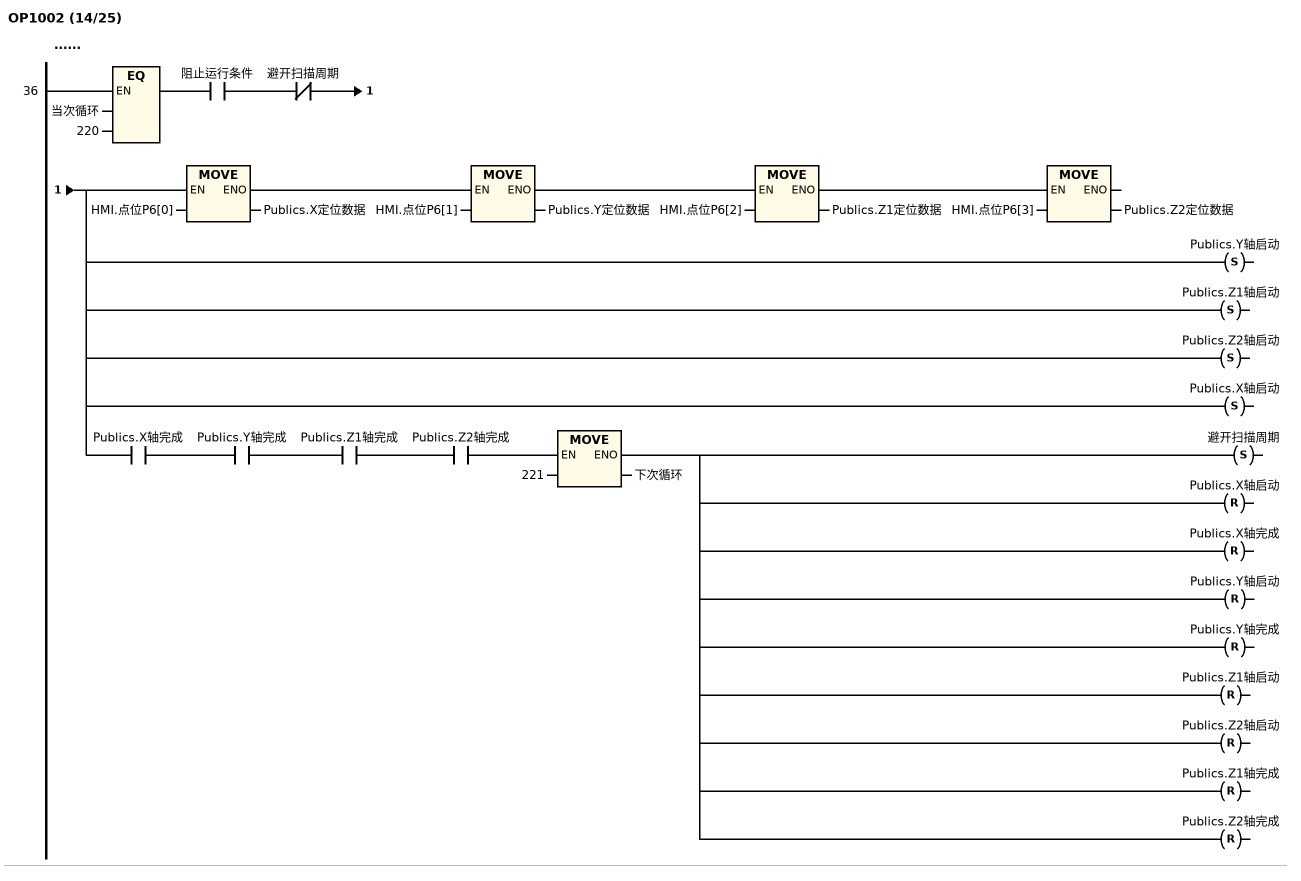
// NETWORK 36: ......
_w44 := 当次循环 = 220 AND 阻止运行条件 AND NOT 避开扫描周期;
IF _w44 THEN Publics.X定位数据 := HMI.点位P6[0]; END_IF
IF _w44 THEN Publics.Y定位数据 := HMI.点位P6[1]; END_IF
IF _w44 THEN Publics.Z1定位数据 := HMI.点位P6[2]; END_IF
IF _w44 THEN Publics.Z2定位数据 := HMI.点位P6[3]; END_IF
Publics.Y轴启动 S= _w44;
Publics.Z1轴启动 S= _w44;
Publics.Z2轴启动 S= _w44;
Publics.X轴启动 S= _w44;
IF _w44 AND Publics.X轴完成 AND Publics.Y轴完成 AND Publics.Z1轴完成 AND Publics.Z2轴完成 THEN 下次循环 := 221; END_IF
_w45 := _w44 AND Publics.X轴完成 AND Publics.Y轴完成 AND Publics.Z1轴完成 AND Publics.Z2轴完成;
避开扫描周期 S= _w45;
Publics.X轴启动 R= _w45;
Publics.X轴完成 R= _w45;
Publics.Y轴启动 R= _w45;
Publics.Y轴完成 R= _w45;
Publics.Z1轴启动 R= _w45;
Publics.Z2轴启动 R= _w45;
Publics.Z1轴完成 R= _w45;
Publics.Z2轴完成 R= _w45;

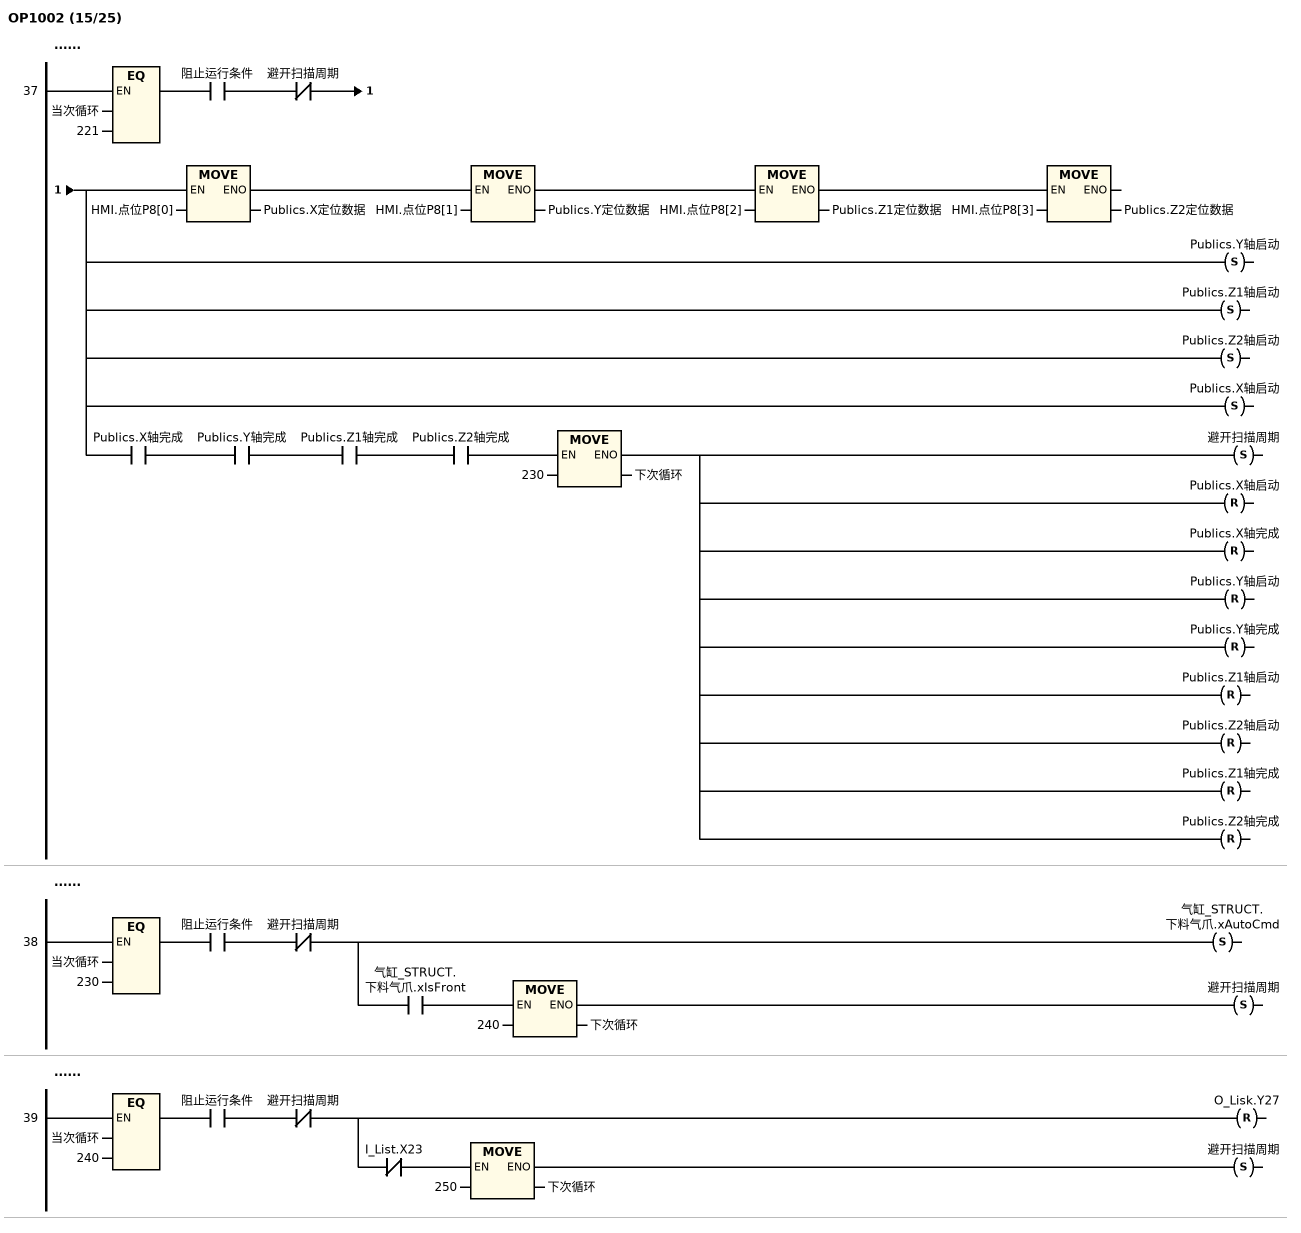
// NETWORK 37: ......
_w46 := 当次循环 = 221 AND 阻止运行条件 AND NOT 避开扫描周期;
IF _w46 THEN Publics.X定位数据 := HMI.点位P8[0]; END_IF
IF _w46 THEN Publics.Y定位数据 := HMI.点位P8[1]; END_IF
IF _w46 THEN Publics.Z1定位数据 := HMI.点位P8[2]; END_IF
IF _w46 THEN Publics.Z2定位数据 := HMI.点位P8[3]; END_IF
Publics.Y轴启动 S= _w46;
Publics.Z1轴启动 S= _w46;
Publics.Z2轴启动 S= _w46;
Publics.X轴启动 S= _w46;
IF _w46 AND Publics.X轴完成 AND Publics.Y轴完成 AND Publics.Z1轴完成 AND Publics.Z2轴完成 THEN 下次循环 := 230; END_IF
_w47 := _w46 AND Publics.X轴完成 AND Publics.Y轴完成 AND Publics.Z1轴完成 AND Publics.Z2轴完成;
避开扫描周期 S= _w47;
Publics.X轴启动 R= _w47;
Publics.X轴完成 R= _w47;
Publics.Y轴启动 R= _w47;
Publics.Y轴完成 R= _w47;
Publics.Z1轴启动 R= _w47;
Publics.Z2轴启动 R= _w47;
Publics.Z1轴完成 R= _w47;
Publics.Z2轴完成 R= _w47;

// NETWORK 38: ......
_w48 := 当次循环 = 230 AND 阻止运行条件 AND NOT 避开扫描周期;
气缸_STRUCT.下料气爪.xAutoCmd S= _w48;
IF _w48 AND 气缸_STRUCT.下料气爪.xIsFront THEN 下次循环 := 240; END_IF
避开扫描周期 S= _w48 AND 气缸_STRUCT.下料气爪.xIsFront;

// NETWORK 39: ......
_w49 := 当次循环 = 240 AND 阻止运行条件 AND NOT 避开扫描周期;
O_Lisk.Y27 R= _w49;
IF _w49 AND NOT I_List.X23 THEN 下次循环 := 250; END_IF
避开扫描周期 S= _w49 AND NOT I_List.X23;

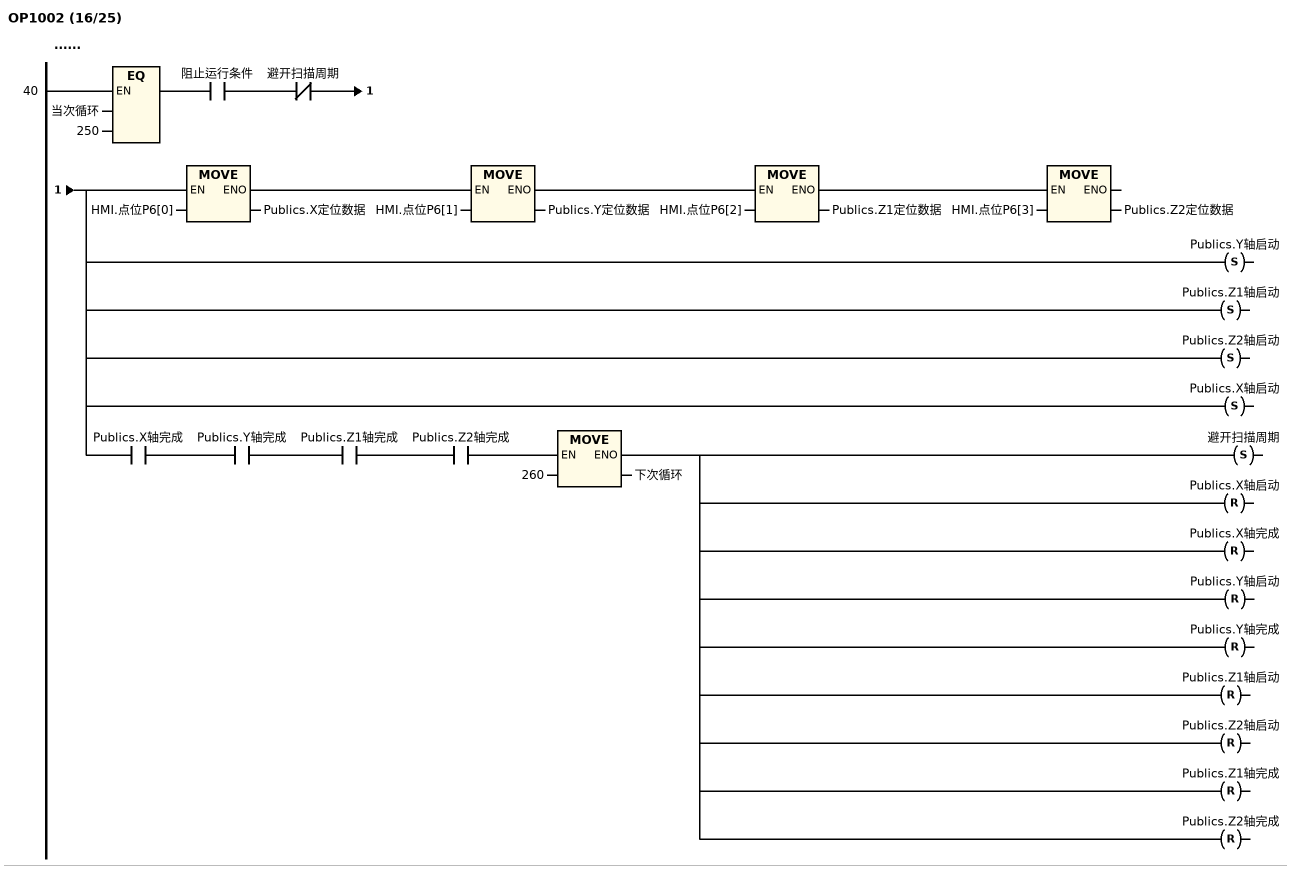
// NETWORK 40: ......
_w50 := 当次循环 = 250 AND 阻止运行条件 AND NOT 避开扫描周期;
IF _w50 THEN Publics.X定位数据 := HMI.点位P6[0]; END_IF
IF _w50 THEN Publics.Y定位数据 := HMI.点位P6[1]; END_IF
IF _w50 THEN Publics.Z1定位数据 := HMI.点位P6[2]; END_IF
IF _w50 THEN Publics.Z2定位数据 := HMI.点位P6[3]; END_IF
Publics.Y轴启动 S= _w50;
Publics.Z1轴启动 S= _w50;
Publics.Z2轴启动 S= _w50;
Publics.X轴启动 S= _w50;
IF _w50 AND Publics.X轴完成 AND Publics.Y轴完成 AND Publics.Z1轴完成 AND Publics.Z2轴完成 THEN 下次循环 := 260; END_IF
_w51 := _w50 AND Publics.X轴完成 AND Publics.Y轴完成 AND Publics.Z1轴完成 AND Publics.Z2轴完成;
避开扫描周期 S= _w51;
Publics.X轴启动 R= _w51;
Publics.X轴完成 R= _w51;
Publics.Y轴启动 R= _w51;
Publics.Y轴完成 R= _w51;
Publics.Z1轴启动 R= _w51;
Publics.Z2轴启动 R= _w51;
Publics.Z1轴完成 R= _w51;
Publics.Z2轴完成 R= _w51;

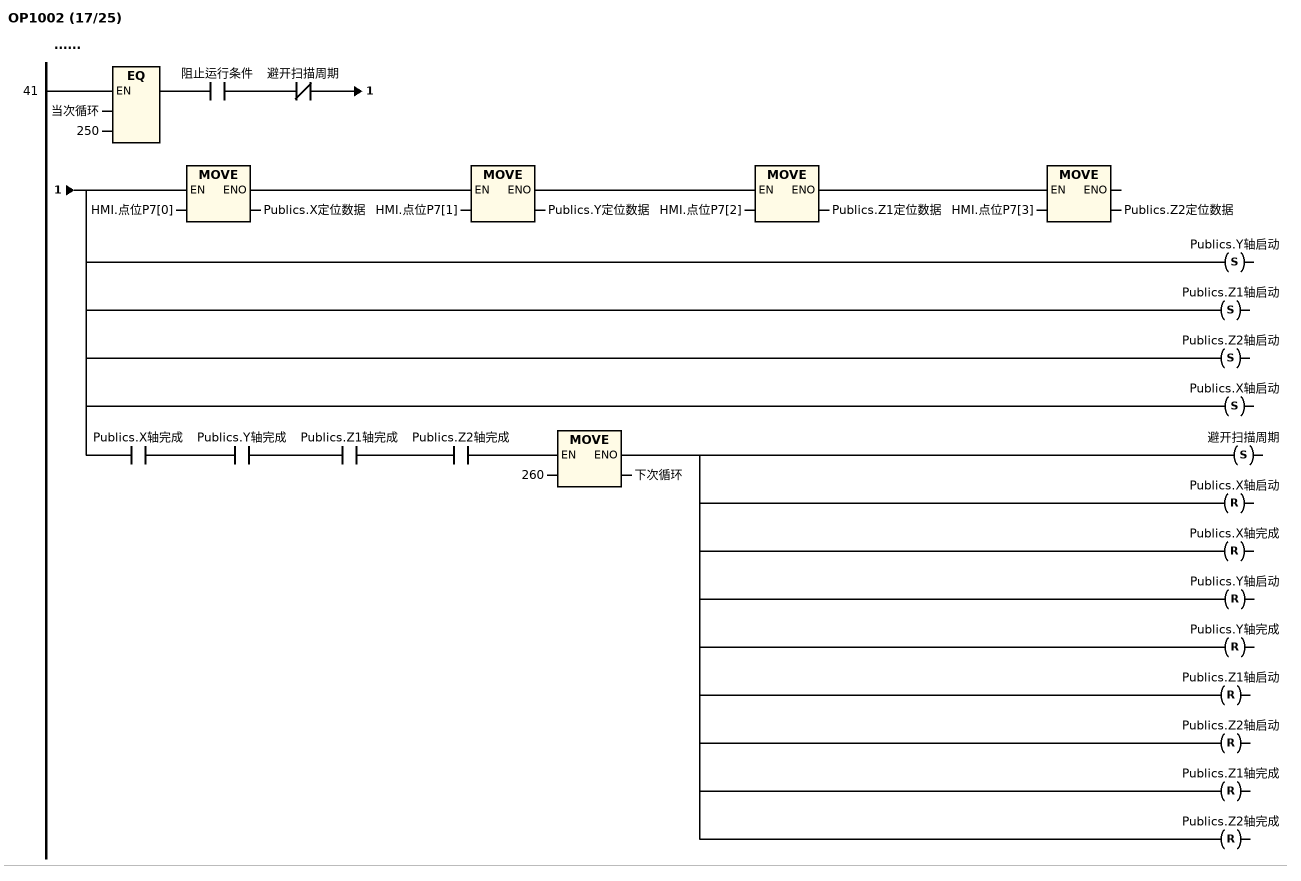
// NETWORK 41: ......
_w52 := 当次循环 = 250 AND 阻止运行条件 AND NOT 避开扫描周期;
IF _w52 THEN Publics.X定位数据 := HMI.点位P7[0]; END_IF
IF _w52 THEN Publics.Y定位数据 := HMI.点位P7[1]; END_IF
IF _w52 THEN Publics.Z1定位数据 := HMI.点位P7[2]; END_IF
IF _w52 THEN Publics.Z2定位数据 := HMI.点位P7[3]; END_IF
Publics.Y轴启动 S= _w52;
Publics.Z1轴启动 S= _w52;
Publics.Z2轴启动 S= _w52;
Publics.X轴启动 S= _w52;
IF _w52 AND Publics.X轴完成 AND Publics.Y轴完成 AND Publics.Z1轴完成 AND Publics.Z2轴完成 THEN 下次循环 := 260; END_IF
_w53 := _w52 AND Publics.X轴完成 AND Publics.Y轴完成 AND Publics.Z1轴完成 AND Publics.Z2轴完成;
避开扫描周期 S= _w53;
Publics.X轴启动 R= _w53;
Publics.X轴完成 R= _w53;
Publics.Y轴启动 R= _w53;
Publics.Y轴完成 R= _w53;
Publics.Z1轴启动 R= _w53;
Publics.Z2轴启动 R= _w53;
Publics.Z1轴完成 R= _w53;
Publics.Z2轴完成 R= _w53;

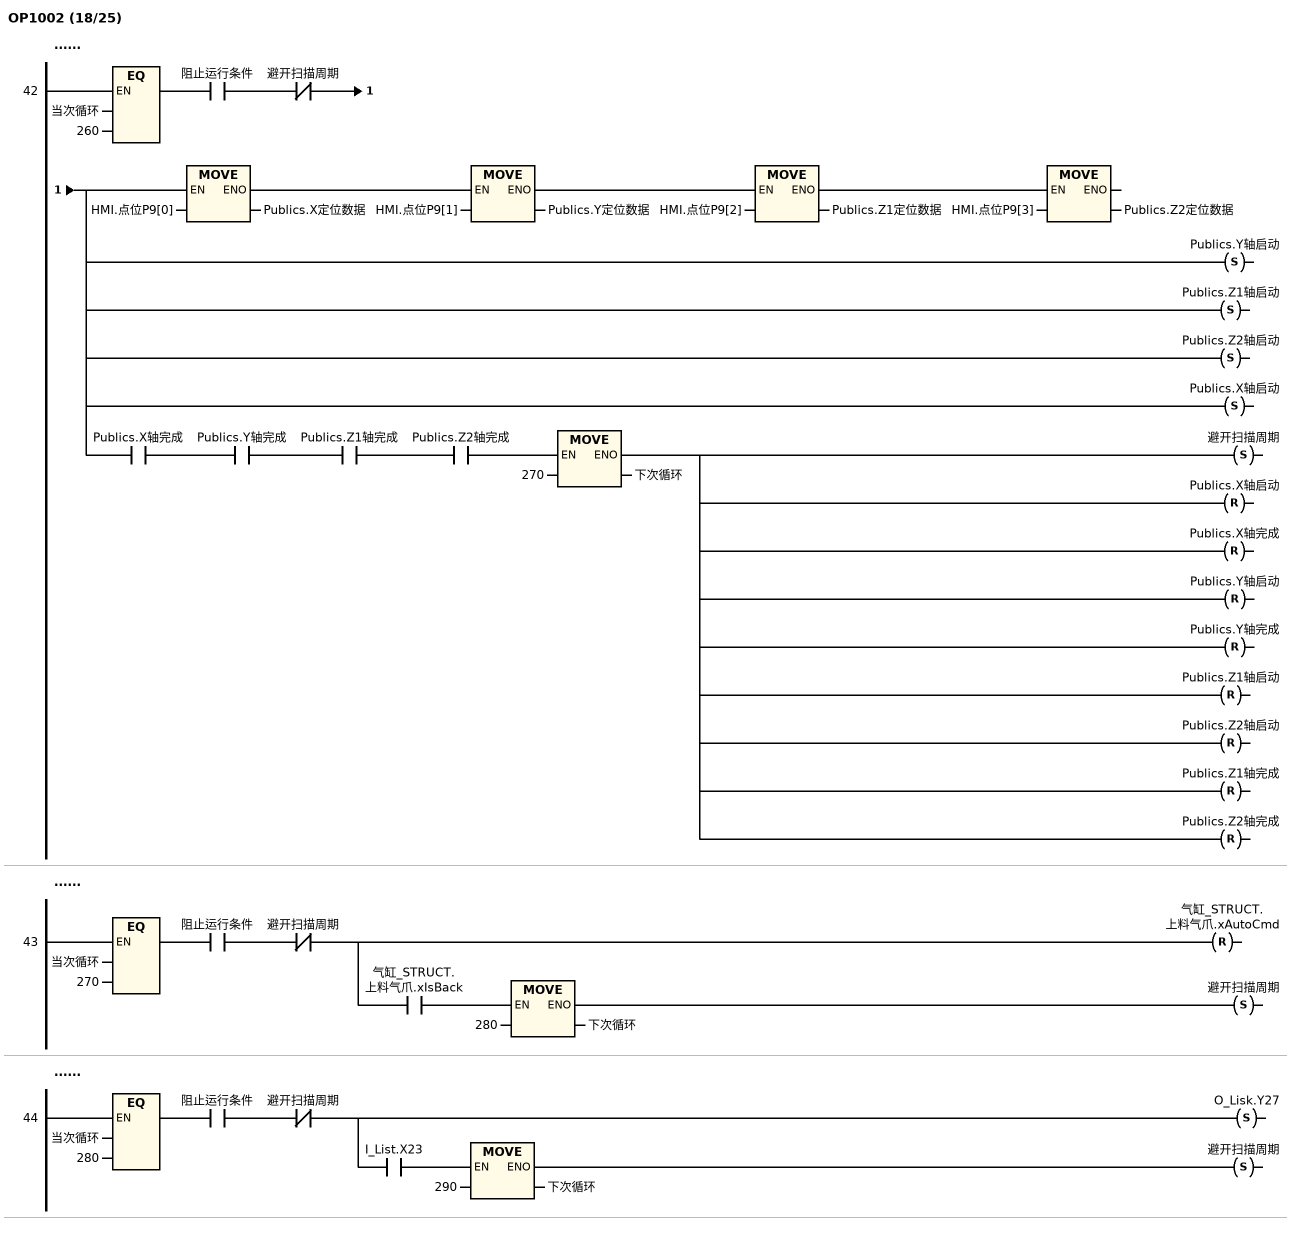
// NETWORK 42: ......
_w54 := 当次循环 = 260 AND 阻止运行条件 AND NOT 避开扫描周期;
IF _w54 THEN Publics.X定位数据 := HMI.点位P9[0]; END_IF
IF _w54 THEN Publics.Y定位数据 := HMI.点位P9[1]; END_IF
IF _w54 THEN Publics.Z1定位数据 := HMI.点位P9[2]; END_IF
IF _w54 THEN Publics.Z2定位数据 := HMI.点位P9[3]; END_IF
Publics.Y轴启动 S= _w54;
Publics.Z1轴启动 S= _w54;
Publics.Z2轴启动 S= _w54;
Publics.X轴启动 S= _w54;
IF _w54 AND Publics.X轴完成 AND Publics.Y轴完成 AND Publics.Z1轴完成 AND Publics.Z2轴完成 THEN 下次循环 := 270; END_IF
_w55 := _w54 AND Publics.X轴完成 AND Publics.Y轴完成 AND Publics.Z1轴完成 AND Publics.Z2轴完成;
避开扫描周期 S= _w55;
Publics.X轴启动 R= _w55;
Publics.X轴完成 R= _w55;
Publics.Y轴启动 R= _w55;
Publics.Y轴完成 R= _w55;
Publics.Z1轴启动 R= _w55;
Publics.Z2轴启动 R= _w55;
Publics.Z1轴完成 R= _w55;
Publics.Z2轴完成 R= _w55;

// NETWORK 43: ......
_w56 := 当次循环 = 270 AND 阻止运行条件 AND NOT 避开扫描周期;
气缸_STRUCT.上料气爪.xAutoCmd R= _w56;
IF _w56 AND 气缸_STRUCT.上料气爪.xIsBack THEN 下次循环 := 280; END_IF
避开扫描周期 S= _w56 AND 气缸_STRUCT.上料气爪.xIsBack;

// NETWORK 44: ......
_w57 := 当次循环 = 280 AND 阻止运行条件 AND NOT 避开扫描周期;
O_Lisk.Y27 S= _w57;
IF _w57 AND I_List.X23 THEN 下次循环 := 290; END_IF
避开扫描周期 S= _w57 AND I_List.X23;

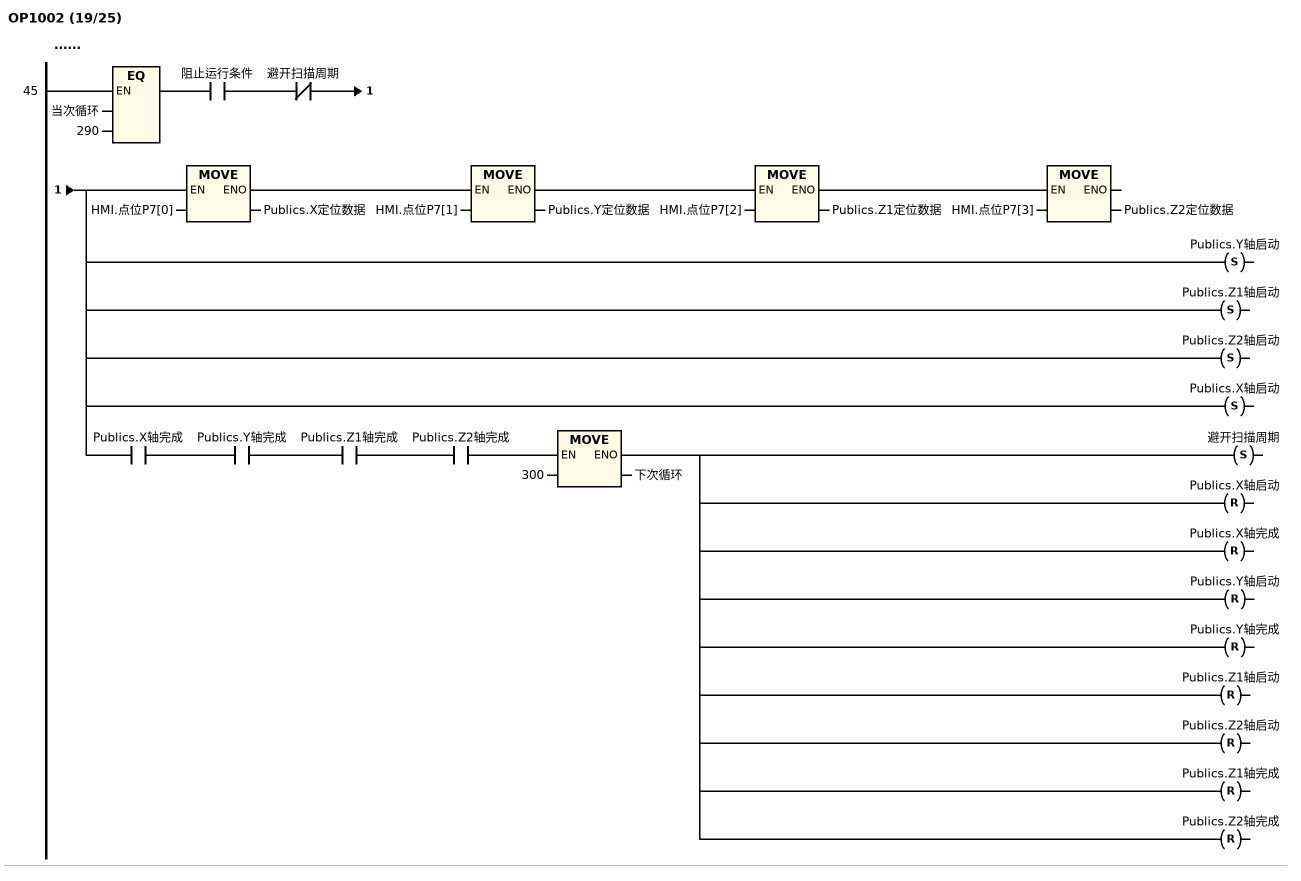
// NETWORK 45: ......
_w58 := 当次循环 = 290 AND 阻止运行条件 AND NOT 避开扫描周期;
IF _w58 THEN Publics.X定位数据 := HMI.点位P7[0]; END_IF
IF _w58 THEN Publics.Y定位数据 := HMI.点位P7[1]; END_IF
IF _w58 THEN Publics.Z1定位数据 := HMI.点位P7[2]; END_IF
IF _w58 THEN Publics.Z2定位数据 := HMI.点位P7[3]; END_IF
Publics.Y轴启动 S= _w58;
Publics.Z1轴启动 S= _w58;
Publics.Z2轴启动 S= _w58;
Publics.X轴启动 S= _w58;
IF _w58 AND Publics.X轴完成 AND Publics.Y轴完成 AND Publics.Z1轴完成 AND Publics.Z2轴完成 THEN 下次循环 := 300; END_IF
_w59 := _w58 AND Publics.X轴完成 AND Publics.Y轴完成 AND Publics.Z1轴完成 AND Publics.Z2轴完成;
避开扫描周期 S= _w59;
Publics.X轴启动 R= _w59;
Publics.X轴完成 R= _w59;
Publics.Y轴启动 R= _w59;
Publics.Y轴完成 R= _w59;
Publics.Z1轴启动 R= _w59;
Publics.Z2轴启动 R= _w59;
Publics.Z1轴完成 R= _w59;
Publics.Z2轴完成 R= _w59;

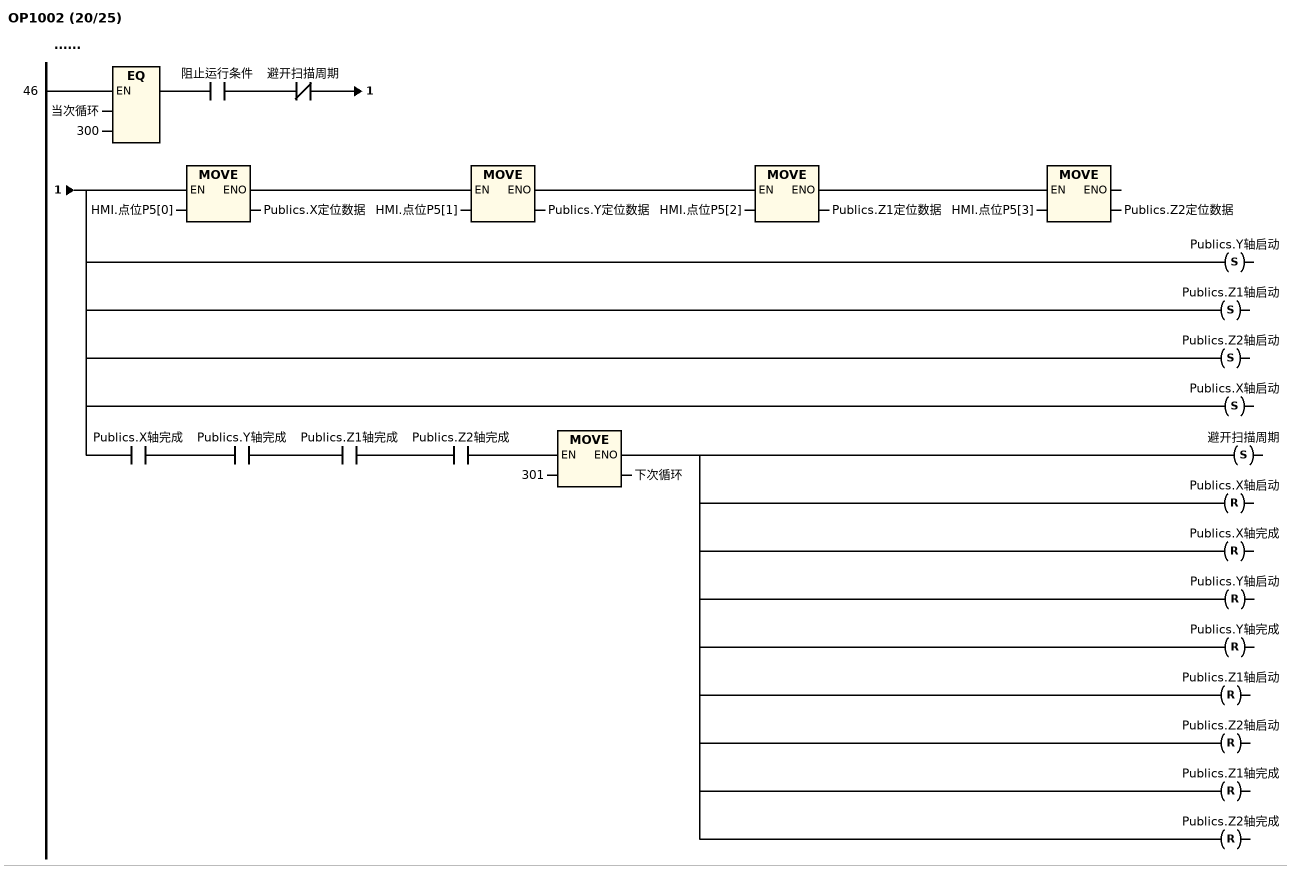
// NETWORK 46: ......
_w60 := 当次循环 = 300 AND 阻止运行条件 AND NOT 避开扫描周期;
IF _w60 THEN Publics.X定位数据 := HMI.点位P5[0]; END_IF
IF _w60 THEN Publics.Y定位数据 := HMI.点位P5[1]; END_IF
IF _w60 THEN Publics.Z1定位数据 := HMI.点位P5[2]; END_IF
IF _w60 THEN Publics.Z2定位数据 := HMI.点位P5[3]; END_IF
Publics.Y轴启动 S= _w60;
Publics.Z1轴启动 S= _w60;
Publics.Z2轴启动 S= _w60;
Publics.X轴启动 S= _w60;
IF _w60 AND Publics.X轴完成 AND Publics.Y轴完成 AND Publics.Z1轴完成 AND Publics.Z2轴完成 THEN 下次循环 := 301; END_IF
_w61 := _w60 AND Publics.X轴完成 AND Publics.Y轴完成 AND Publics.Z1轴完成 AND Publics.Z2轴完成;
避开扫描周期 S= _w61;
Publics.X轴启动 R= _w61;
Publics.X轴完成 R= _w61;
Publics.Y轴启动 R= _w61;
Publics.Y轴完成 R= _w61;
Publics.Z1轴启动 R= _w61;
Publics.Z2轴启动 R= _w61;
Publics.Z1轴完成 R= _w61;
Publics.Z2轴完成 R= _w61;

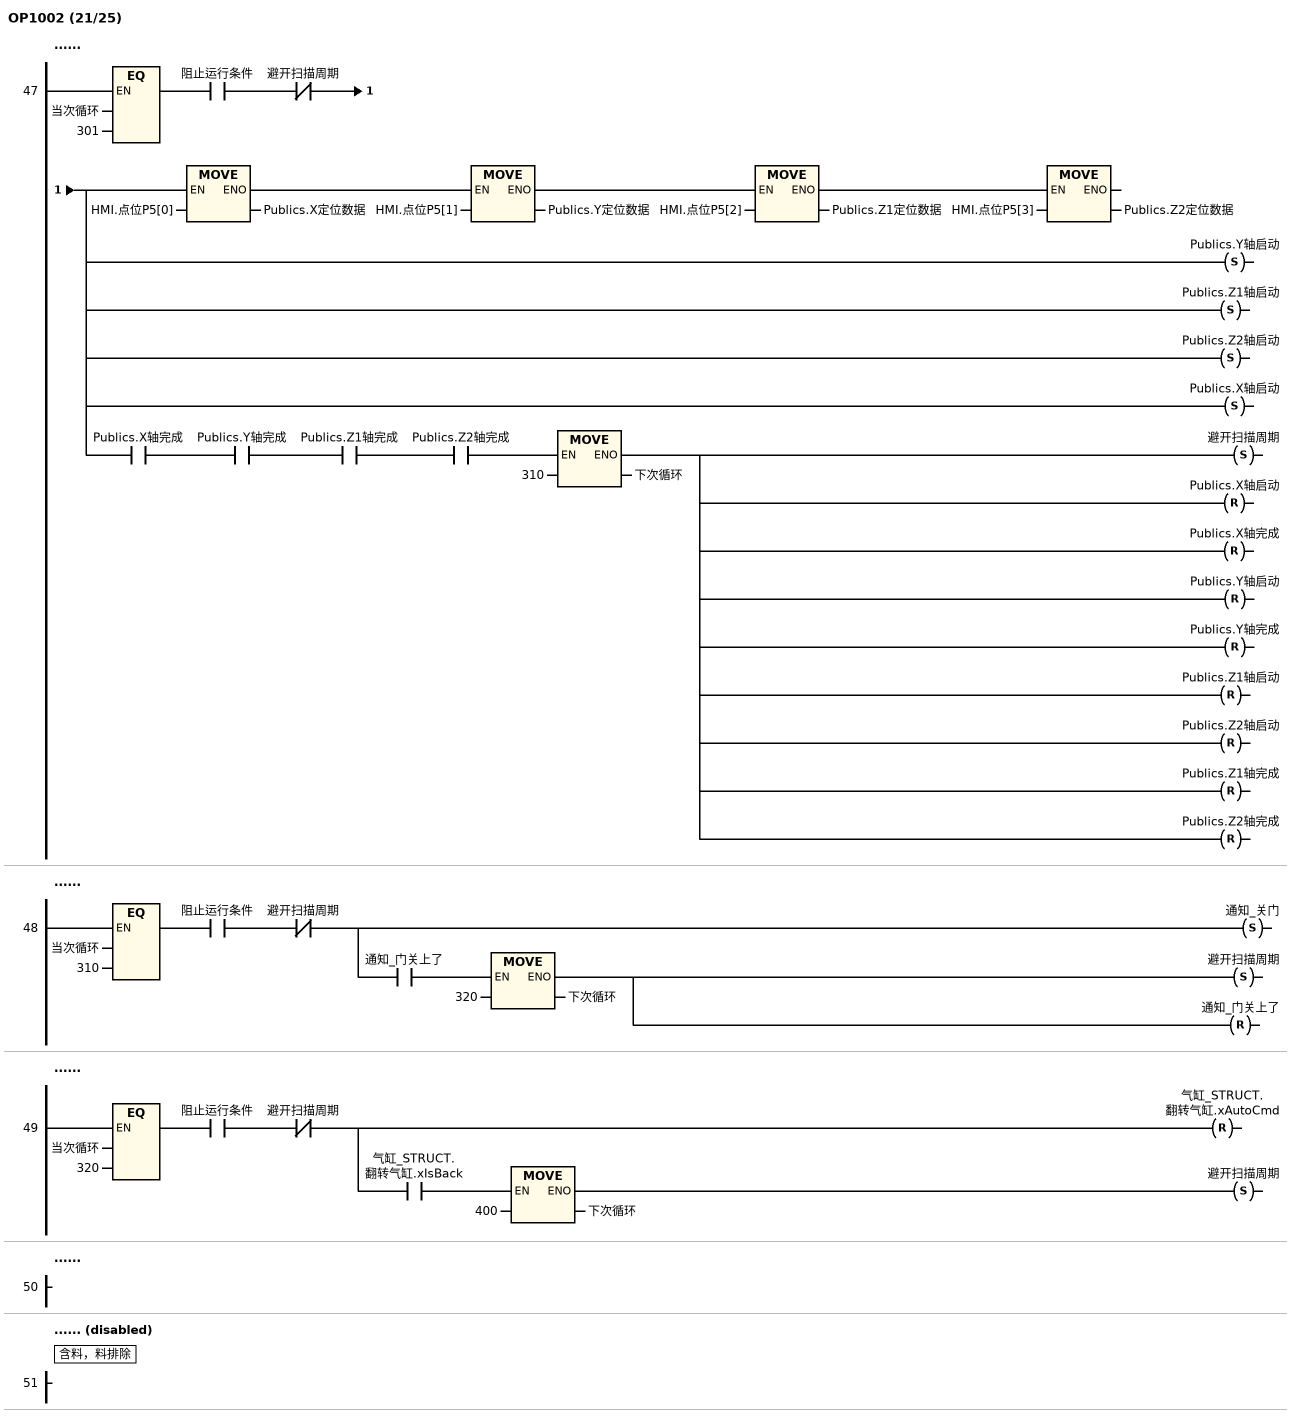
// NETWORK 47: ......
_w62 := 当次循环 = 301 AND 阻止运行条件 AND NOT 避开扫描周期;
IF _w62 THEN Publics.X定位数据 := HMI.点位P5[0]; END_IF
IF _w62 THEN Publics.Y定位数据 := HMI.点位P5[1]; END_IF
IF _w62 THEN Publics.Z1定位数据 := HMI.点位P5[2]; END_IF
IF _w62 THEN Publics.Z2定位数据 := HMI.点位P5[3]; END_IF
Publics.Y轴启动 S= _w62;
Publics.Z1轴启动 S= _w62;
Publics.Z2轴启动 S= _w62;
Publics.X轴启动 S= _w62;
IF _w62 AND Publics.X轴完成 AND Publics.Y轴完成 AND Publics.Z1轴完成 AND Publics.Z2轴完成 THEN 下次循环 := 310; END_IF
_w63 := _w62 AND Publics.X轴完成 AND Publics.Y轴完成 AND Publics.Z1轴完成 AND Publics.Z2轴完成;
避开扫描周期 S= _w63;
Publics.X轴启动 R= _w63;
Publics.X轴完成 R= _w63;
Publics.Y轴启动 R= _w63;
Publics.Y轴完成 R= _w63;
Publics.Z1轴启动 R= _w63;
Publics.Z2轴启动 R= _w63;
Publics.Z1轴完成 R= _w63;
Publics.Z2轴完成 R= _w63;

// NETWORK 48: ......
_w64 := 当次循环 = 310 AND 阻止运行条件 AND NOT 避开扫描周期;
通知_关门 S= _w64;
IF _w64 AND 通知_门关上了 THEN 下次循环 := 320; END_IF
_w65 := _w64 AND 通知_门关上了;
避开扫描周期 S= _w65;
通知_门关上了 R= _w65;

// NETWORK 49: ......
_w66 := 当次循环 = 320 AND 阻止运行条件 AND NOT 避开扫描周期;
气缸_STRUCT.翻转气缸.xAutoCmd R= _w66;
IF _w66 AND 气缸_STRUCT.翻转气缸.xIsBack THEN 下次循环 := 400; END_IF
避开扫描周期 S= _w66 AND 气缸_STRUCT.翻转气缸.xIsBack;

// NETWORK 50: ......

// NETWORK 51: ...... (disabled)
// label: 含料，料排除

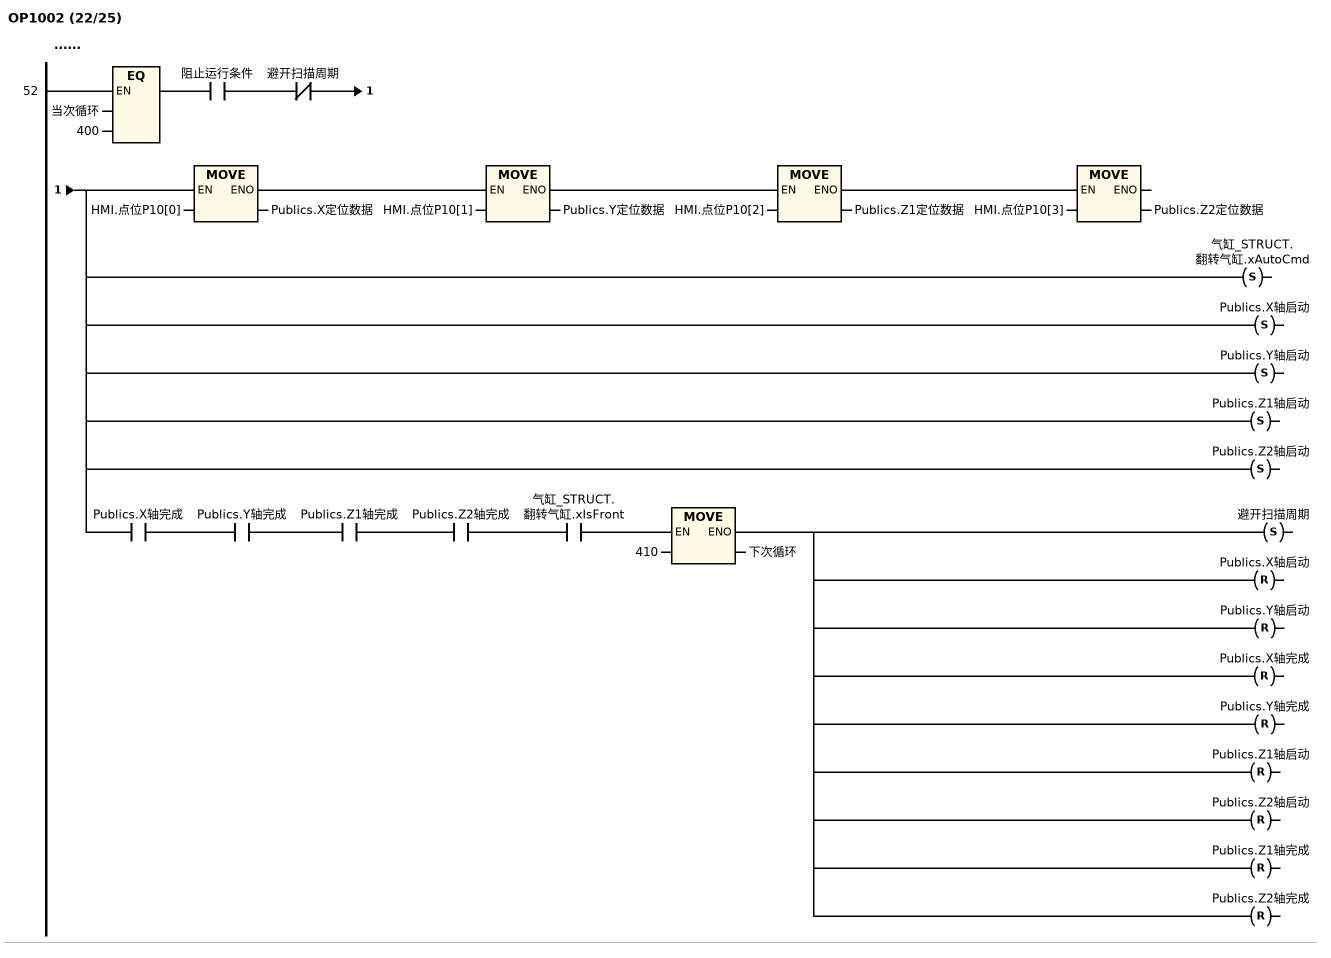
// NETWORK 52: ......
_w67 := 当次循环 = 400 AND 阻止运行条件 AND NOT 避开扫描周期;
IF _w67 THEN Publics.X定位数据 := HMI.点位P10[0]; END_IF
IF _w67 THEN Publics.Y定位数据 := HMI.点位P10[1]; END_IF
IF _w67 THEN Publics.Z1定位数据 := HMI.点位P10[2]; END_IF
IF _w67 THEN Publics.Z2定位数据 := HMI.点位P10[3]; END_IF
气缸_STRUCT.翻转气缸.xAutoCmd S= _w67;
Publics.X轴启动 S= _w67;
Publics.Y轴启动 S= _w67;
Publics.Z1轴启动 S= _w67;
Publics.Z2轴启动 S= _w67;
IF _w67 AND Publics.X轴完成 AND Publics.Y轴完成 AND Publics.Z1轴完成 AND Publics.Z2轴完成 AND 气缸_STRUCT.翻转气缸.xIsFront THEN
    下次循环 := 410;
END_IF
_w68 := _w67 AND Publics.X轴完成 AND Publics.Y轴完成 AND Publics.Z1轴完成 AND Publics.Z2轴完成 AND 气缸_STRUCT.翻转气缸.xIsFront;
避开扫描周期 S= _w68;
Publics.X轴启动 R= _w68;
Publics.Y轴启动 R= _w68;
Publics.X轴完成 R= _w68;
Publics.Y轴完成 R= _w68;
Publics.Z1轴启动 R= _w68;
Publics.Z2轴启动 R= _w68;
Publics.Z1轴完成 R= _w68;
Publics.Z2轴完成 R= _w68;

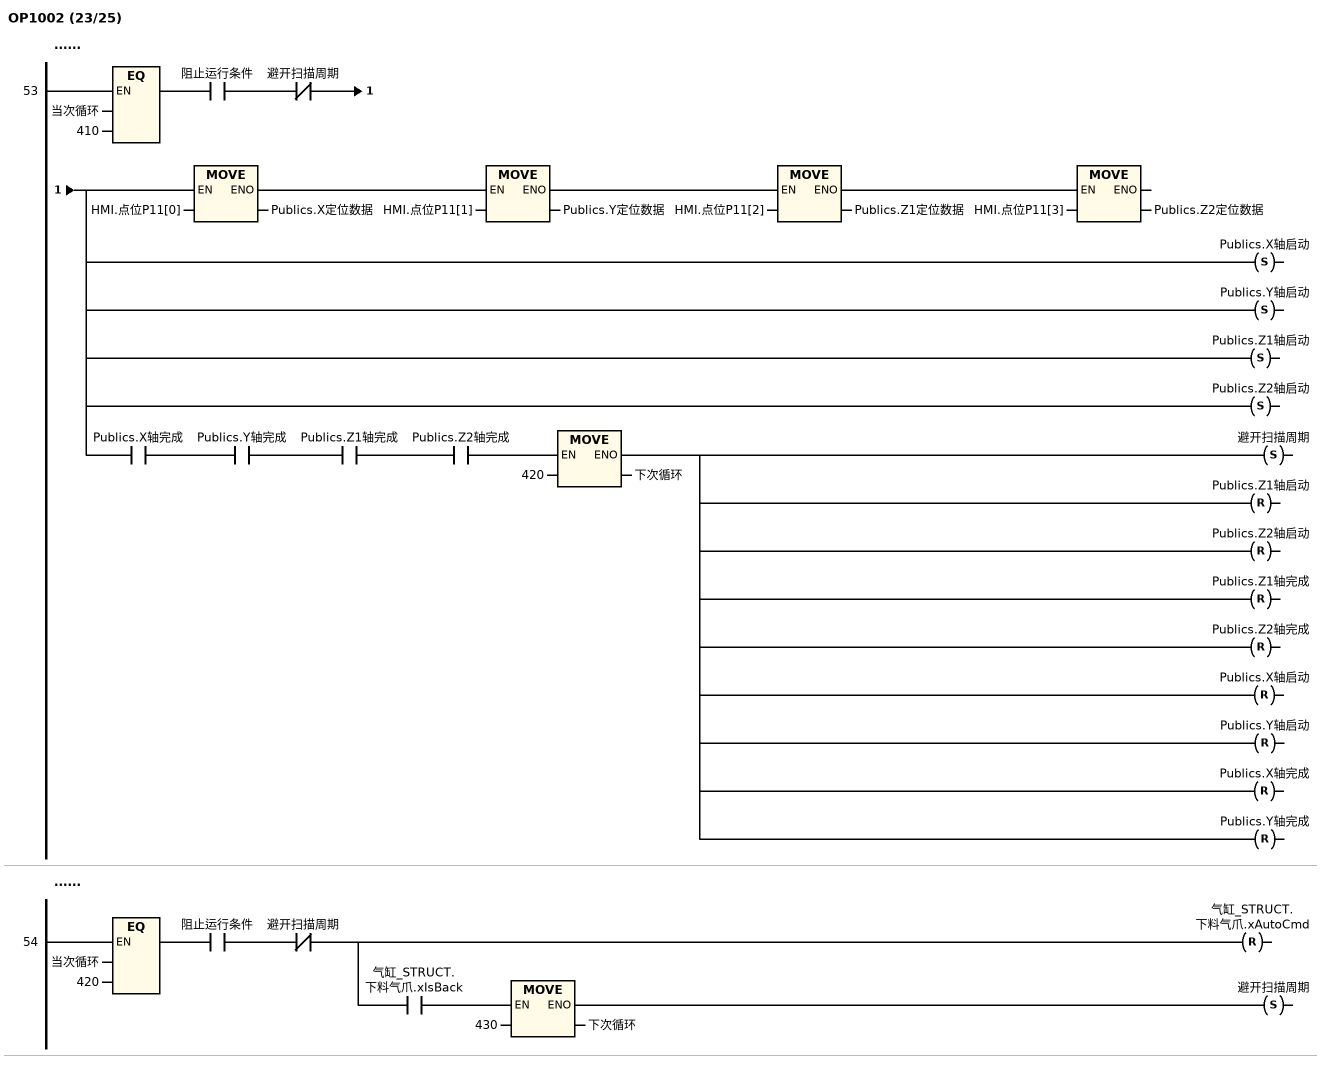
// NETWORK 53: ......
_w69 := 当次循环 = 410 AND 阻止运行条件 AND NOT 避开扫描周期;
IF _w69 THEN Publics.X定位数据 := HMI.点位P11[0]; END_IF
IF _w69 THEN Publics.Y定位数据 := HMI.点位P11[1]; END_IF
IF _w69 THEN Publics.Z1定位数据 := HMI.点位P11[2]; END_IF
IF _w69 THEN Publics.Z2定位数据 := HMI.点位P11[3]; END_IF
Publics.X轴启动 S= _w69;
Publics.Y轴启动 S= _w69;
Publics.Z1轴启动 S= _w69;
Publics.Z2轴启动 S= _w69;
IF _w69 AND Publics.X轴完成 AND Publics.Y轴完成 AND Publics.Z1轴完成 AND Publics.Z2轴完成 THEN 下次循环 := 420; END_IF
_w70 := _w69 AND Publics.X轴完成 AND Publics.Y轴完成 AND Publics.Z1轴完成 AND Publics.Z2轴完成;
避开扫描周期 S= _w70;
Publics.Z1轴启动 R= _w70;
Publics.Z2轴启动 R= _w70;
Publics.Z1轴完成 R= _w70;
Publics.Z2轴完成 R= _w70;
Publics.X轴启动 R= _w70;
Publics.Y轴启动 R= _w70;
Publics.X轴完成 R= _w70;
Publics.Y轴完成 R= _w70;

// NETWORK 54: ......
_w71 := 当次循环 = 420 AND 阻止运行条件 AND NOT 避开扫描周期;
气缸_STRUCT.下料气爪.xAutoCmd R= _w71;
IF _w71 AND 气缸_STRUCT.下料气爪.xIsBack THEN 下次循环 := 430; END_IF
避开扫描周期 S= _w71 AND 气缸_STRUCT.下料气爪.xIsBack;

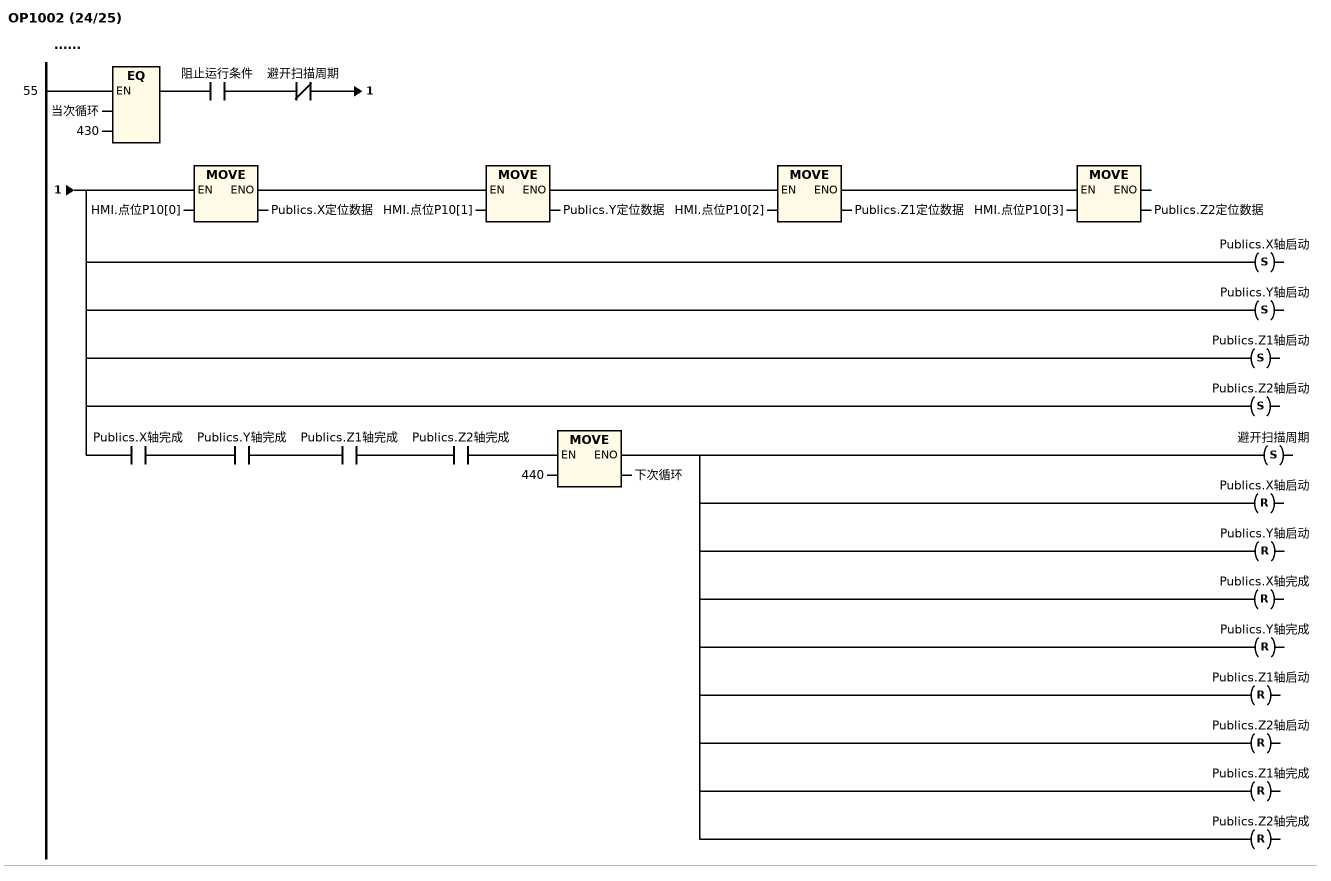
// NETWORK 55: ......
_w72 := 当次循环 = 430 AND 阻止运行条件 AND NOT 避开扫描周期;
IF _w72 THEN Publics.X定位数据 := HMI.点位P10[0]; END_IF
IF _w72 THEN Publics.Y定位数据 := HMI.点位P10[1]; END_IF
IF _w72 THEN Publics.Z1定位数据 := HMI.点位P10[2]; END_IF
IF _w72 THEN Publics.Z2定位数据 := HMI.点位P10[3]; END_IF
Publics.X轴启动 S= _w72;
Publics.Y轴启动 S= _w72;
Publics.Z1轴启动 S= _w72;
Publics.Z2轴启动 S= _w72;
IF _w72 AND Publics.X轴完成 AND Publics.Y轴完成 AND Publics.Z1轴完成 AND Publics.Z2轴完成 THEN 下次循环 := 440; END_IF
_w73 := _w72 AND Publics.X轴完成 AND Publics.Y轴完成 AND Publics.Z1轴完成 AND Publics.Z2轴完成;
避开扫描周期 S= _w73;
Publics.X轴启动 R= _w73;
Publics.Y轴启动 R= _w73;
Publics.X轴完成 R= _w73;
Publics.Y轴完成 R= _w73;
Publics.Z1轴启动 R= _w73;
Publics.Z2轴启动 R= _w73;
Publics.Z1轴完成 R= _w73;
Publics.Z2轴完成 R= _w73;

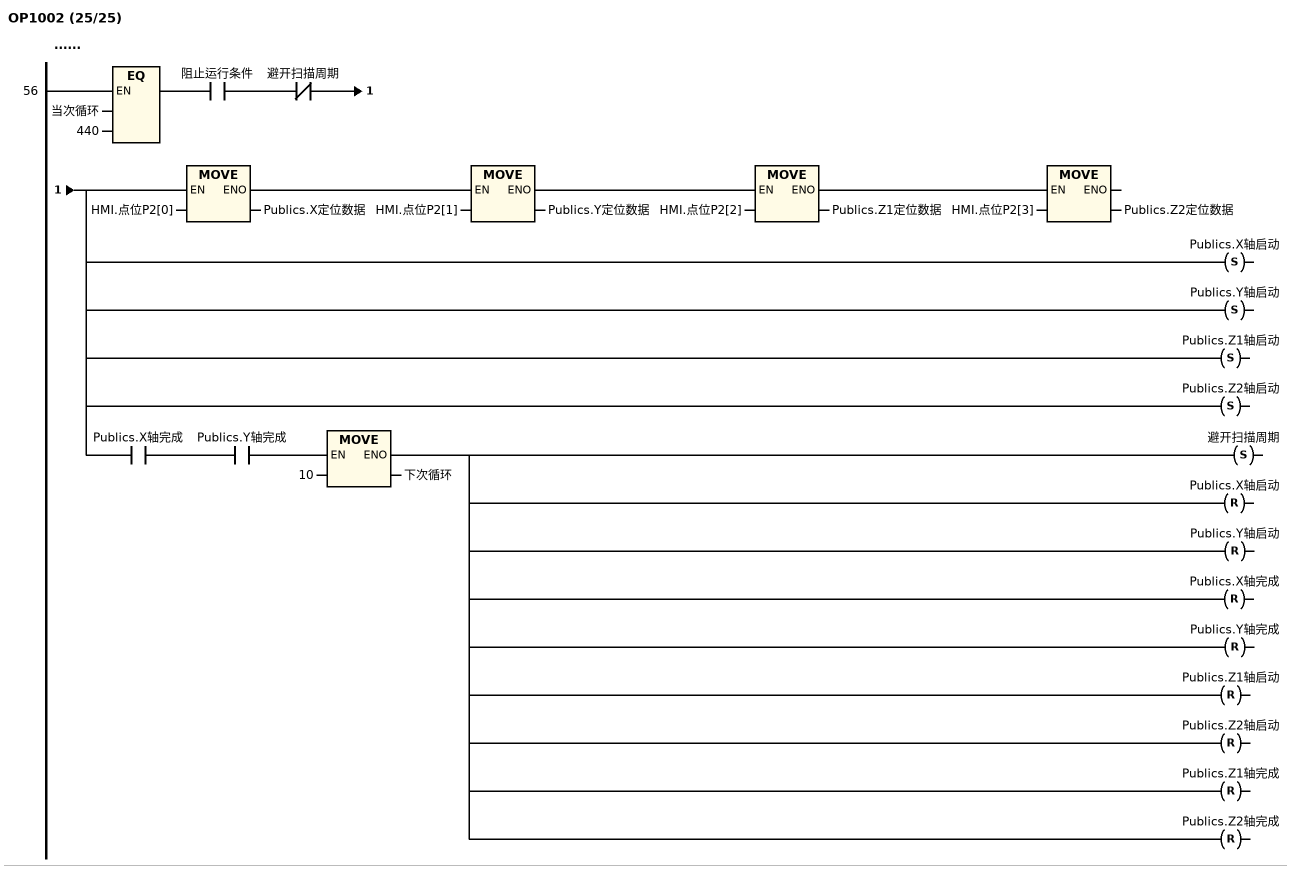
// NETWORK 56: ......
_w74 := 当次循环 = 440 AND 阻止运行条件 AND NOT 避开扫描周期;
IF _w74 THEN Publics.X定位数据 := HMI.点位P2[0]; END_IF
IF _w74 THEN Publics.Y定位数据 := HMI.点位P2[1]; END_IF
IF _w74 THEN Publics.Z1定位数据 := HMI.点位P2[2]; END_IF
IF _w74 THEN Publics.Z2定位数据 := HMI.点位P2[3]; END_IF
Publics.X轴启动 S= _w74;
Publics.Y轴启动 S= _w74;
Publics.Z1轴启动 S= _w74;
Publics.Z2轴启动 S= _w74;
IF _w74 AND Publics.X轴完成 AND Publics.Y轴完成 THEN 下次循环 := 10; END_IF
_w75 := _w74 AND Publics.X轴完成 AND Publics.Y轴完成;
避开扫描周期 S= _w75;
Publics.X轴启动 R= _w75;
Publics.Y轴启动 R= _w75;
Publics.X轴完成 R= _w75;
Publics.Y轴完成 R= _w75;
Publics.Z1轴启动 R= _w75;
Publics.Z2轴启动 R= _w75;
Publics.Z1轴完成 R= _w75;
Publics.Z2轴完成 R= _w75;

ACTION 辅助流程:
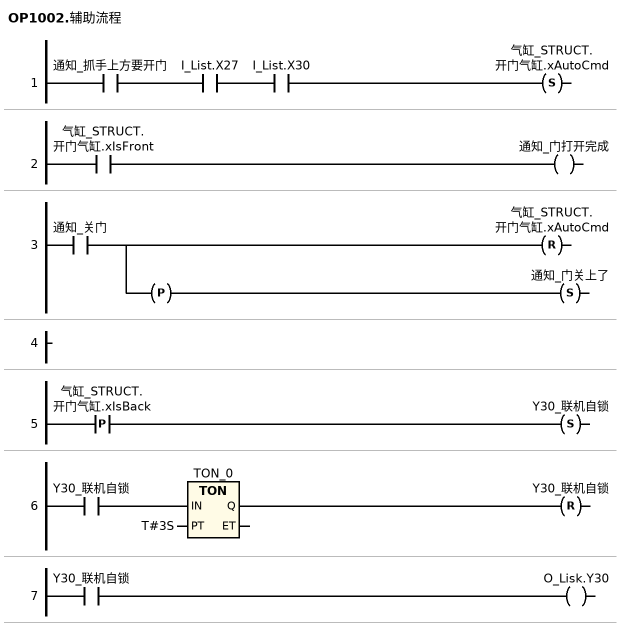
// NETWORK 1
气缸_STRUCT.开门气缸.xAutoCmd S= 通知_抓手上方要开门 AND I_List.X27 AND I_List.X30;

// NETWORK 2
通知_门打开完成 := 气缸_STRUCT.开门气缸.xIsFront;

// NETWORK 3
气缸_STRUCT.开门气缸.xAutoCmd R= 通知_关门;
_rt2(CLK := 通知_关门);
通知_门关上了 S= _rt2.Q;

// NETWORK 4

// NETWORK 5
_rt3(CLK := 气缸_STRUCT.开门气缸.xIsBack);
Y30_联机自锁 S= _rt3.Q;

// NETWORK 6
TON_0(IN := Y30_联机自锁, PT := T#3S); // TON
Y30_联机自锁 R= TON_0.Q;

// NETWORK 7
O_Lisk.Y30 := Y30_联机自锁;
END_ACTION

END_PROGRAM

// Device/Application/气缸
PROGRAM 气缸
VAR
	FB_CylinderSingle_0: FB_CylinderSingle;
	上料推出气缸到位延时: word;
	上料推出气缸原位延时: word;
	FB_CylinderSingle_1: FB_CylinderSingle;
	上料推出气缸报警复位: BOOL;
	上料顶起气缸原位延时: WORD;
	上料顶起气缸到位位延时: WORD;
	FB_CylinderSingle_2: FB_CylinderSingle;
	FB_CylinderSingle_3: FB_CylinderSingle;
	FB_CylinderSingle_4: FB_CylinderSingle;
	FB_CylinderSingle_5: FB_CylinderSingle;
	FB_CylinderSingle_6: FB_CylinderSingle;
	A1: BOOL;
	A2: BOOL;
	A3: BOOL;
	A4: BOOL;
	A5: BOOL;
	A6: BOOL;
END_VAR

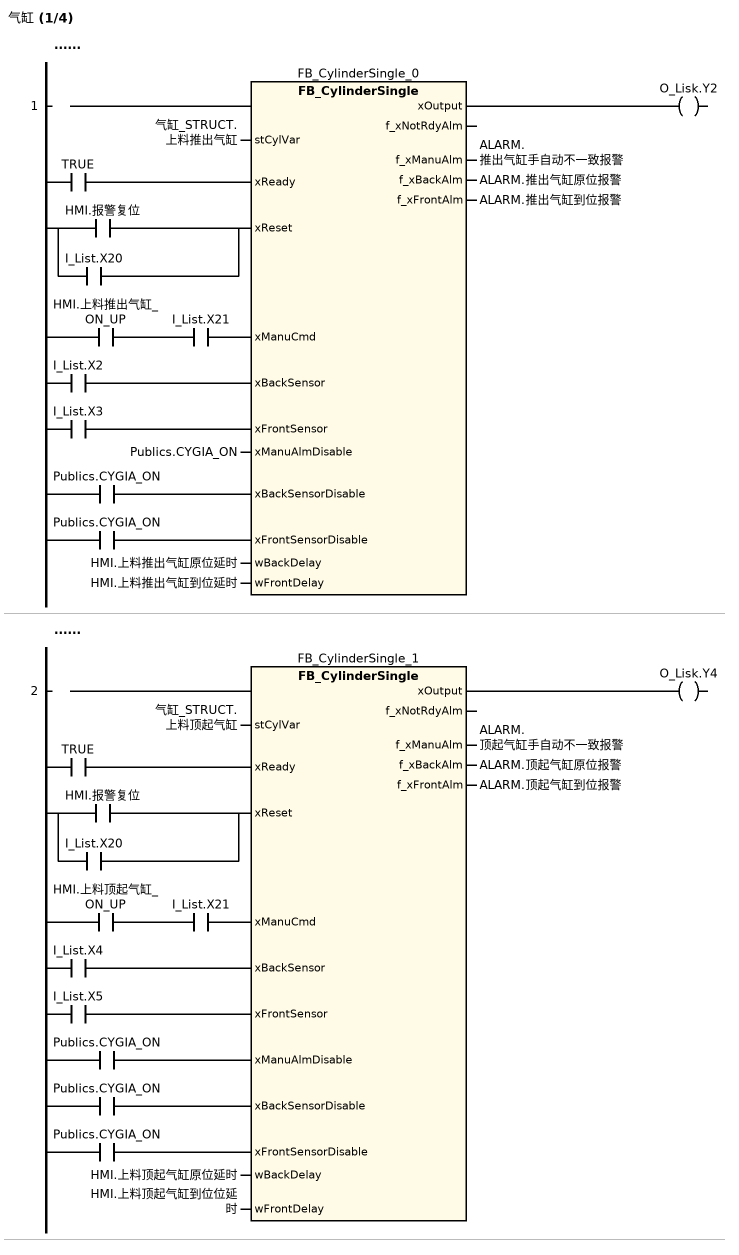
// NETWORK 1: ......
FB_CylinderSingle_0(
    stCylVar := 气缸_STRUCT.上料推出气缸,
    xReady := TRUE,
    xReset := HMI.报警复位 OR I_List.X20,
    xManuCmd := HMI.上料推出气缸_ON_UP AND I_List.X21,
    xBackSensor := I_List.X2,
    xFrontSensor := I_List.X3,
    xManuAlmDisable := Publics.CYGIA_ON,
    xBackSensorDisable := Publics.CYGIA_ON,
    xFrontSensorDisable := Publics.CYGIA_ON,
    wBackDelay := HMI.上料推出气缸原位延时,
    wFrontDelay := HMI.上料推出气缸到位延时,
    f_xManuAlm => ALARM.推出气缸手自动不一致报警,
    f_xBackAlm => ALARM.推出气缸原位报警,
    f_xFrontAlm => ALARM.推出气缸到位报警); // FB_CylinderSingle
O_Lisk.Y2 := FB_CylinderSingle_0.xOutput;

// NETWORK 2: ......
FB_CylinderSingle_1(
    stCylVar := 气缸_STRUCT.上料顶起气缸,
    xReady := TRUE,
    xReset := HMI.报警复位 OR I_List.X20,
    xManuCmd := HMI.上料顶起气缸_ON_UP AND I_List.X21,
    xBackSensor := I_List.X4,
    xFrontSensor := I_List.X5,
    xManuAlmDisable := Publics.CYGIA_ON,
    xBackSensorDisable := Publics.CYGIA_ON,
    xFrontSensorDisable := Publics.CYGIA_ON,
    wBackDelay := HMI.上料顶起气缸原位延时,
    wFrontDelay := HMI.上料顶起气缸到位位延时,
    f_xManuAlm => ALARM.顶起气缸手自动不一致报警,
    f_xBackAlm => ALARM.顶起气缸原位报警,
    f_xFrontAlm => ALARM.顶起气缸到位报警); // FB_CylinderSingle
O_Lisk.Y4 := FB_CylinderSingle_1.xOutput;

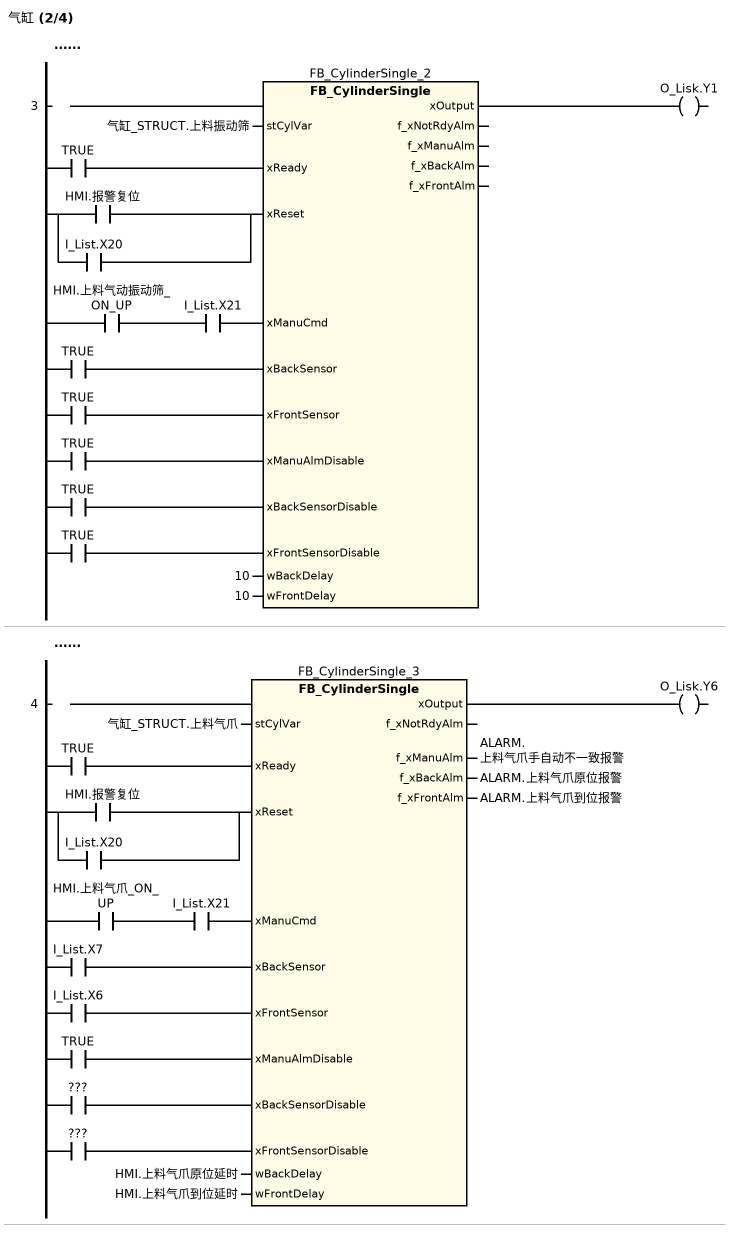
// NETWORK 3: ......
FB_CylinderSingle_2(
    stCylVar := 气缸_STRUCT.上料振动筛,
    xReady := TRUE,
    xReset := HMI.报警复位 OR I_List.X20,
    xManuCmd := HMI.上料气动振动筛_ON_UP AND I_List.X21,
    xBackSensor := TRUE,
    xFrontSensor := TRUE,
    xManuAlmDisable := TRUE,
    xBackSensorDisable := TRUE,
    xFrontSensorDisable := TRUE,
    wBackDelay := 10,
    wFrontDelay := 10); // FB_CylinderSingle
O_Lisk.Y1 := FB_CylinderSingle_2.xOutput;

// NETWORK 4: ......
FB_CylinderSingle_3(
    stCylVar := 气缸_STRUCT.上料气爪,
    xReady := TRUE,
    xReset := HMI.报警复位 OR I_List.X20,
    xManuCmd := HMI.上料气爪_ON_UP AND I_List.X21,
    xBackSensor := I_List.X7,
    xFrontSensor := I_List.X6,
    xManuAlmDisable := TRUE,
    wBackDelay := HMI.上料气爪原位延时,
    wFrontDelay := HMI.上料气爪到位延时,
    f_xManuAlm => ALARM.上料气爪手自动不一致报警,
    f_xBackAlm => ALARM.上料气爪原位报警,
    f_xFrontAlm => ALARM.上料气爪到位报警); // FB_CylinderSingle
O_Lisk.Y6 := FB_CylinderSingle_3.xOutput;

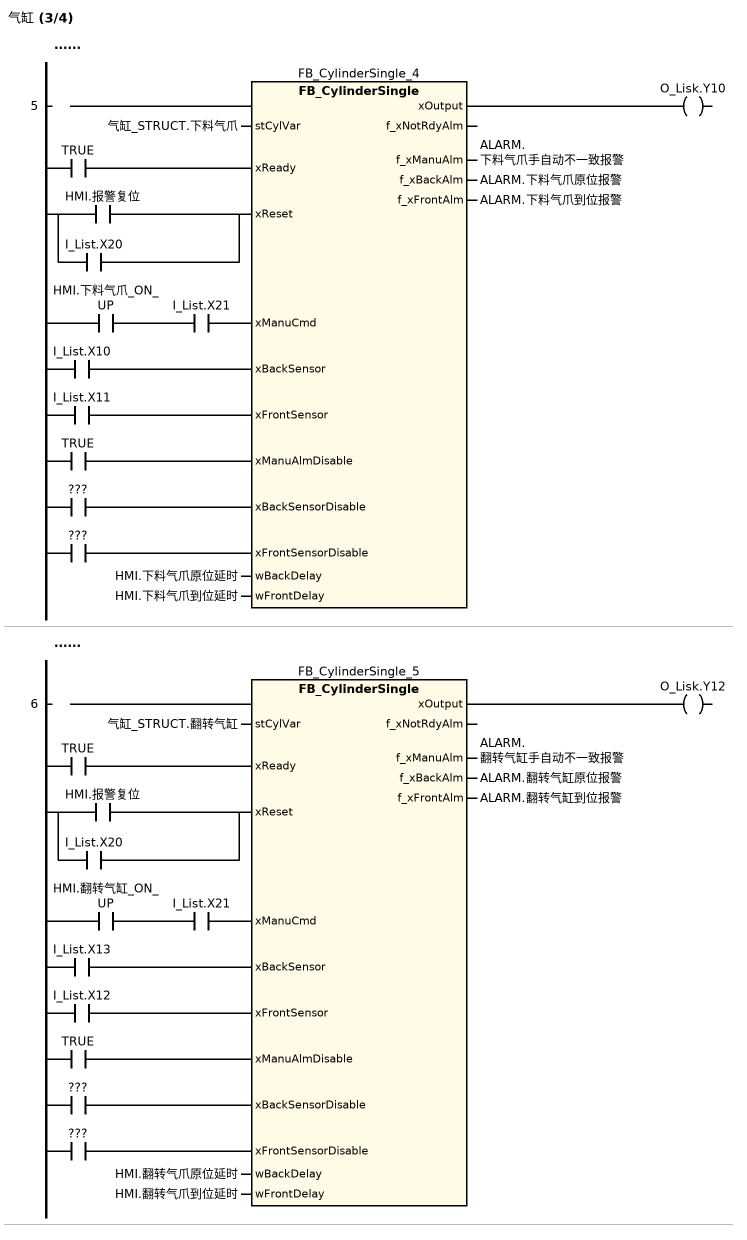
// NETWORK 5: ......
FB_CylinderSingle_4(
    stCylVar := 气缸_STRUCT.下料气爪,
    xReady := TRUE,
    xReset := HMI.报警复位 OR I_List.X20,
    xManuCmd := HMI.下料气爪_ON_UP AND I_List.X21,
    xBackSensor := I_List.X10,
    xFrontSensor := I_List.X11,
    xManuAlmDisable := TRUE,
    wBackDelay := HMI.下料气爪原位延时,
    wFrontDelay := HMI.下料气爪到位延时,
    f_xManuAlm => ALARM.下料气爪手自动不一致报警,
    f_xBackAlm => ALARM.下料气爪原位报警,
    f_xFrontAlm => ALARM.下料气爪到位报警); // FB_CylinderSingle
O_Lisk.Y10 := FB_CylinderSingle_4.xOutput;

// NETWORK 6: ......
FB_CylinderSingle_5(
    stCylVar := 气缸_STRUCT.翻转气缸,
    xReady := TRUE,
    xReset := HMI.报警复位 OR I_List.X20,
    xManuCmd := HMI.翻转气缸_ON_UP AND I_List.X21,
    xBackSensor := I_List.X13,
    xFrontSensor := I_List.X12,
    xManuAlmDisable := TRUE,
    wBackDelay := HMI.翻转气爪原位延时,
    wFrontDelay := HMI.翻转气爪到位延时,
    f_xManuAlm => ALARM.翻转气缸手自动不一致报警,
    f_xBackAlm => ALARM.翻转气缸原位报警,
    f_xFrontAlm => ALARM.翻转气缸到位报警); // FB_CylinderSingle
O_Lisk.Y12 := FB_CylinderSingle_5.xOutput;

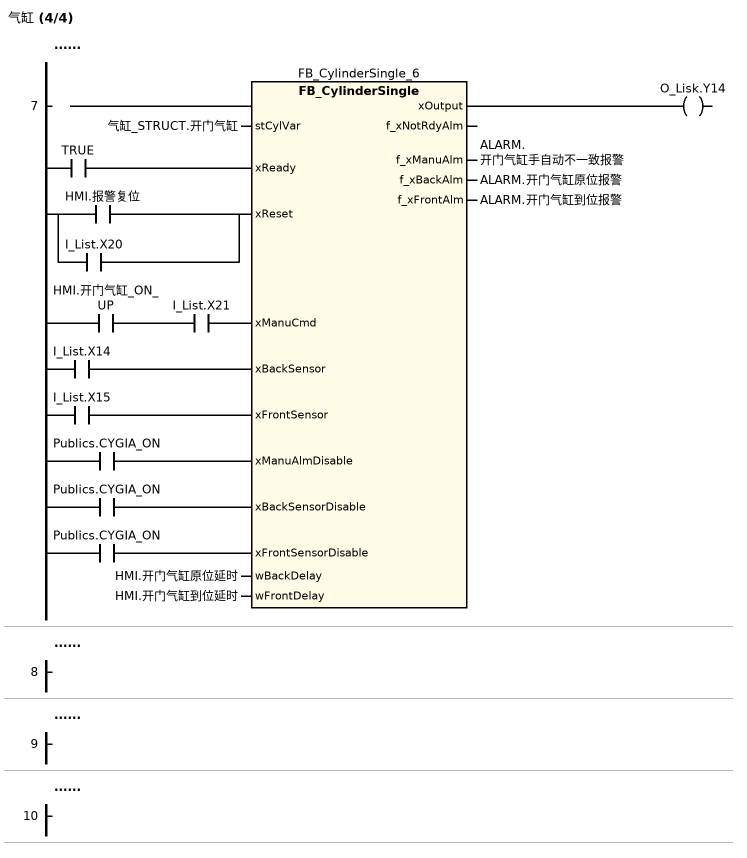
// NETWORK 7: ......
FB_CylinderSingle_6(
    stCylVar := 气缸_STRUCT.开门气缸,
    xReady := TRUE,
    xReset := HMI.报警复位 OR I_List.X20,
    xManuCmd := HMI.开门气缸_ON_UP AND I_List.X21,
    xBackSensor := I_List.X14,
    xFrontSensor := I_List.X15,
    xManuAlmDisable := Publics.CYGIA_ON,
    xBackSensorDisable := Publics.CYGIA_ON,
    xFrontSensorDisable := Publics.CYGIA_ON,
    wBackDelay := HMI.开门气缸原位延时,
    wFrontDelay := HMI.开门气缸到位延时,
    f_xManuAlm => ALARM.开门气缸手自动不一致报警,
    f_xBackAlm => ALARM.开门气缸原位报警,
    f_xFrontAlm => ALARM.开门气缸到位报警); // FB_CylinderSingle
O_Lisk.Y14 := FB_CylinderSingle_6.xOutput;

// NETWORK 8: ......

// NETWORK 9: ......

// NETWORK 10: ......

END_PROGRAM

// Device/Application/FunctionBlock/FB_CylinderSingle
FUNCTION_BLOCK FB_CylinderSingle
VAR_IN_OUT
	stCylVar: CYLINDER_REF;
END_VAR
VAR_INPUT
	///安全条件
	xReady: BOOL;
	///报警复位
	xReset: BOOL;
	///手动控制,每on一次,则反转输出点状态
	xManuCmd: BOOL;
	///原位检测
	xBackSensor: BOOL;
	///到位检测
	xFrontSensor: BOOL;
	///手自动不一致报警无效
	xManuAlmDisable: BOOL;
	///原位检测无效
	xBackSensorDisable: BOOL;
	///到位检测无效
	xFrontSensorDisable: BOOL;
	///原位延时
	wBackDelay: WORD;
	///到位延时
	wFrontDelay: WORD;
END_VAR
VAR_OUTPUT
	xOutput: BOOL;
	///未满足安全条件报警
	f_xNotRdyAlm: BOOL;
	///手自动不一致报警	
	f_xManuAlm: BOOL;
	///未在原位报警
	f_xBackAlm: BOOL;
	///未到位报警
	f_xFrontAlm: BOOL;
END_VAR
VAR
	///获取自动控制的上升沿
	fbAutoRise: R_TRIG;
	///获取自动控制的下升沿
	fbAutoFall: F_TRIG;
	///获取手动控制的下升沿
	fbManuFall: F_TRIG;
	///获取复位信号的上升沿
	fbResetRise: R_TRIG;
	///原位状态延时,用于输出原位状态
	fbBackTon: TON;
	///到位状态延时,用于输出到位状态
	fbFrontTon: TON;
	///获取原位状态下降沿	
	fbBackFall: F_TRIG;
	///获取到位状态下降沿
	fbFrontFall: F_TRIG;
	///原位动作超时,用于输出未在原位位置报警
	fbBackWait: TON;
	///到位动作超时,用于输出未在到位位置报警
	fbFrontWait: TON;
END_VAR

   //初始化时复位输出点
   IF xReady AND stCylVar.xInit AND ( NOT f_xNotRdyAlm	) THEN
	    xOutput := FALSE;
	    f_xManuAlm  := FALSE;
	    stCylVar.xInit  := FALSE;
 
   END_IF


   //获取手动控制、自动控制的边沿信号
   fbManuFall(CLK:=xManuCmd , Q=> );
   fbAutoRise(CLK:=stCylvar.xAutoCmd , Q=> );
   fbAutoFall(CLK:=stCylvar.xAutoCmd , Q=> );
      
    //1,手动操作时，如果满足安全条件且未屏蔽了手自动不一致报警时，则输出点反转，  
    IF xReady AND (NOT xManuAlmDisable) AND fbManuFall.Q THEN
   	    xOutput  := NOT xOutput ;
		//手动操作生效时，判断输出点状态与自动命令是否一致，不一致时,置位手动操作执行中报警；一致时复位该报警。
	    //当因安全条件不满足导致自动命令未执行时，可通过手动操作控制其动作执行,此时手动操作并不引起手动操作执行中报警。
		 IF ( stCylvar.xAutoCmd ) XOR xOutput THEN
   	   	    f_xManuAlm  :=TRUE;
   	     ELSE 
   	   	    f_xManuAlm  :=FALSE;
   	     END_IF  	 	
     END_IF
	 
	//2,手动操作时，如果满足安全条件且屏蔽了手自动不一致报警时，则自动控制点反转、复位手自动不一致报警，  
    IF xReady AND  xManuAlmDisable AND fbManuFall.Q THEN
   	    stCylvar.xAutoCmd  := NOT stCylvar.xAutoCmd ;
		f_xManuAlm  :=FALSE;		  	 	
    END_IF
   
   
   
   //自动命令置位时，如果满足安全条件，则输出点置位
   IF xReady AND fbAutoRise.Q THEN
   	   xOutput  :=TRUE;
   END_IF
      
   //自动命令复位时，如满足安全条件，则输出点复位。
   IF xReady AND fbAutoFall.Q THEN
   	    xOutput  :=FALSE;		
   END_IF
   
   
   //原位状态输出
   fbBackTon(IN:= ( NOT xOutput) AND ( NOT xFrontSensor ) AND ( xBackSensor OR xBackSensorDisable ) , PT:= WORD_TO_TIME ( wBackDelay *10 ) , Q=> stCylvar.xIsBack, ET=> );
   
   
   //到位状态输出
   fbFrontTon(IN:= xOutput AND ( xFrontSensor OR xFrontSensorDisable ) AND ( NOT xBackSensor ) , PT:= WORD_TO_TIME ( wFrontDelay *10 ), Q=> stCylvar.xIsFront, ET=> );
      
	  
   //报警复位
   fbResetRise(CLK:= xReset, Q=> );
   IF fbResetRise.Q THEN
   	   f_xNotRdyAlm := FALSE;
	   f_xFrontAlm := FALSE;
	   f_xBackAlm := FALSE;
   
   END_IF
   
   
   //未满足安全条件报警
   //当手动操作或自动命令状态发生改变时，如果不能满足安全条件，则输出未满足安全条件报警
   IF ( fbManuFall.Q OR fbAutoRise.Q OR fbAutoFall.Q ) AND ( NOT xReady ) THEN
   	    f_xNotRdyAlm := TRUE; 
   END_IF
   
   
   //未在原位报警
   //自动命令变OFF后(上电后气缸处于自由状态时不判断)，延时5秒，如果原位标志未变为ON、且未发生手动操作和安全条件报警，则输出未到原位报警
   fbBackWait(IN:=  NOT stCylvar.xAutoCmd  , PT:= T#5S , Q=> , ET=> );
   fbBackFall(CLK:= stCylvar.xIsBack , Q=> );
   IF (( fbBackWait.Q AND (NOT stCylvar.xIsBack )) OR (( NOT stCylvar.xAutoCmd ) AND fbBackFall.Q )) AND  ( NOT f_xManuAlm ) AND  ( NOT f_xNotRdyAlm ) THEN
   	    f_xBackAlm := TRUE;
   END_IF
   
   
   //未到位报警
   //自动命令变ON后，延时5秒，如果到位标志未变为ON、且未发生手动操作和安全条件报警，则输出未到位报警
   fbFrontWait(IN:= stCylvar.xAutoCmd , PT:= T#5S , Q=> , ET=> );
   fbFrontFall(CLK:= stCylvar.xIsFront, Q=> );
   IF ( ( fbFrontWait.Q AND ( NOT stCylvar.xIsFront ) ) OR (stCylvar.xAutoCmd AND fbFrontFall.Q )) AND ( NOT f_xManuAlm ) AND ( NOT f_xNotRdyAlm ) THEN
   	    f_xFrontAlm := TRUE;   
   END_IF

END_FUNCTION_BLOCK

// Device/Application/Servo_Ctrol
PROGRAM Servo_Ctrol
VAR
	总线复位: BOOL;
	SMC3_ReinitDrive_0: SMC3_ReinitDrive;
	SMC3_ReinitDrive_1: SMC3_ReinitDrive;
	SMC3_ReinitDrive_2: SMC3_ReinitDrive;
	SMC3_ReinitDrive_3: SMC3_ReinitDrive;
	Y轴_使能: MC_Power;
	Z2轴_使能: MC_Power;
	Z1轴_使能: MC_Power;
	X轴_使能: MC_Power;
	MC_Jog_0: MC_Jog;
	Y轴_JOG: MC_Jog;
	Z2轴_JOG: MC_Jog;
	Z1轴_JOG: MC_Jog;
	X轴_JOG: MC_Jog;
	AXIS3: AXIS_REF_SM3;
	MC_Reset_0: MC_Reset;
	MC_Reset_1: MC_Reset;
	MC_Reset_2: MC_Reset;
	MC_Reset_3: MC_Reset;
	MC_ReadStatus_0: MC_ReadStatus;
	MC_ReadAxisError_0: MC_ReadAxisError;
	MC_ReadActualPosition_0: MC_ReadActualPosition;
	MC_ReadActualPosition_1: MC_ReadActualPosition;
	MC_ReadActualPosition_2: MC_ReadActualPosition;
	MC_ReadActualPosition_3: MC_ReadActualPosition;
	MC_Halt_0: MC_Halt;
	MC_Halt_1: MC_Halt;
	MC_Halt_2: MC_Halt;
	MC_Halt_3: MC_Halt;
	MC_Stop_0: MC_Stop;
	MC_Stop_1: MC_Stop;
	MC_Stop_2: MC_Stop;
	MC_Stop_3: MC_Stop;
	Z2定位: MC_MoveAbsolute;
	Z1定位: MC_MoveAbsolute;
	Y定位: MC_MoveAbsolute;
	X定位: MC_MoveAbsolute;
	MC_Home_0: MC_Home;
	MC_Home_1: MC_Home;
	MC_Home_2: MC_Home;
	MC_Home_3: MC_Home;
END_VAR
VAR // added by the converter: edge detectors and wires of the graphical bodies
    _rt1, _rt2, _rt3, _rt4, _rt5, _rt6, _rt7 : R_TRIG;
END_VAR

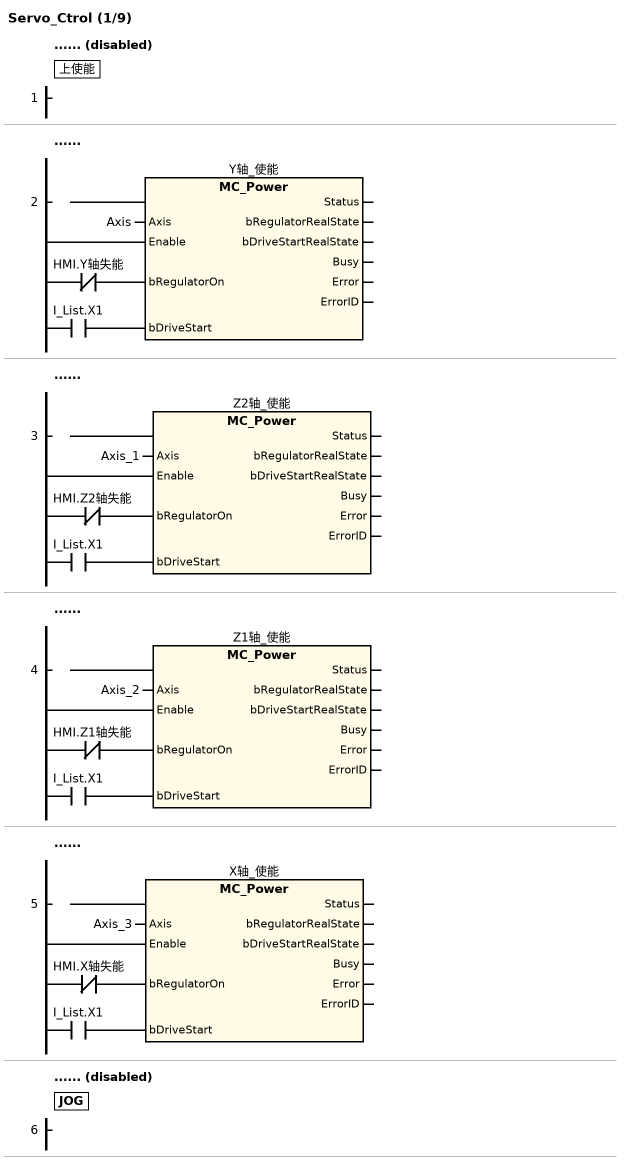
// NETWORK 1: ...... (disabled)
// label: 上使能

// NETWORK 2: ......
Y轴_使能(Axis := Axis, Enable := TRUE, bRegulatorOn := NOT HMI.Y轴失能, bDriveStart := I_List.X1); // MC_Power

// NETWORK 3: ......
Z2轴_使能(Axis := Axis_1, Enable := TRUE, bRegulatorOn := NOT HMI.Z2轴失能, bDriveStart := I_List.X1); // MC_Power

// NETWORK 4: ......
Z1轴_使能(Axis := Axis_2, Enable := TRUE, bRegulatorOn := NOT HMI.Z1轴失能, bDriveStart := I_List.X1); // MC_Power

// NETWORK 5: ......
X轴_使能(Axis := Axis_3, Enable := TRUE, bRegulatorOn := NOT HMI.X轴失能, bDriveStart := I_List.X1); // MC_Power

// NETWORK 6: ...... (disabled)
// label: JOG

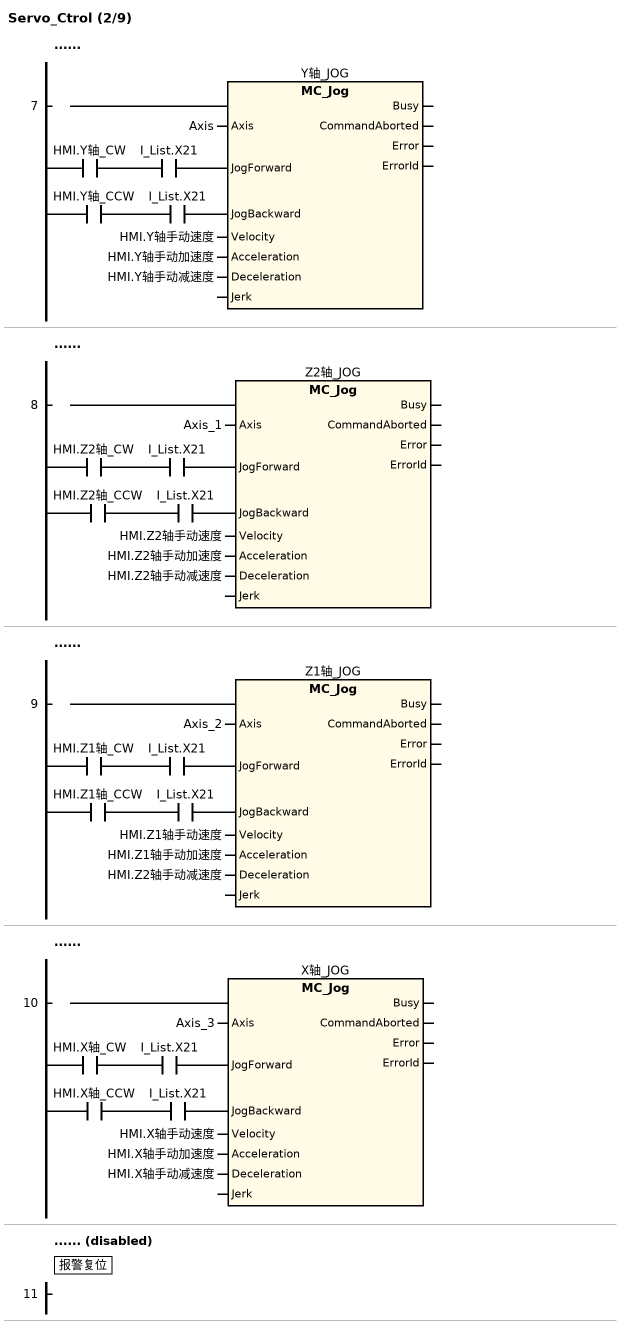
// NETWORK 7: ......
Y轴_JOG(
    Axis := Axis,
    JogForward := HMI.Y轴_CW AND I_List.X21,
    JogBackward := HMI.Y轴_CCW AND I_List.X21,
    Velocity := HMI.Y轴手动速度,
    Acceleration := HMI.Y轴手动加速度,
    Deceleration := HMI.Y轴手动减速度); // MC_Jog

// NETWORK 8: ......
Z2轴_JOG(
    Axis := Axis_1,
    JogForward := HMI.Z2轴_CW AND I_List.X21,
    JogBackward := HMI.Z2轴_CCW AND I_List.X21,
    Velocity := HMI.Z2轴手动速度,
    Acceleration := HMI.Z2轴手动加速度,
    Deceleration := HMI.Z2轴手动减速度); // MC_Jog

// NETWORK 9: ......
Z1轴_JOG(
    Axis := Axis_2,
    JogForward := HMI.Z1轴_CW AND I_List.X21,
    JogBackward := HMI.Z1轴_CCW AND I_List.X21,
    Velocity := HMI.Z1轴手动速度,
    Acceleration := HMI.Z1轴手动加速度,
    Deceleration := HMI.Z2轴手动减速度); // MC_Jog

// NETWORK 10: ......
X轴_JOG(
    Axis := Axis_3,
    JogForward := HMI.X轴_CW AND I_List.X21,
    JogBackward := HMI.X轴_CCW AND I_List.X21,
    Velocity := HMI.X轴手动速度,
    Acceleration := HMI.X轴手动加速度,
    Deceleration := HMI.X轴手动减速度); // MC_Jog

// NETWORK 11: ...... (disabled)
// label: 报警复位

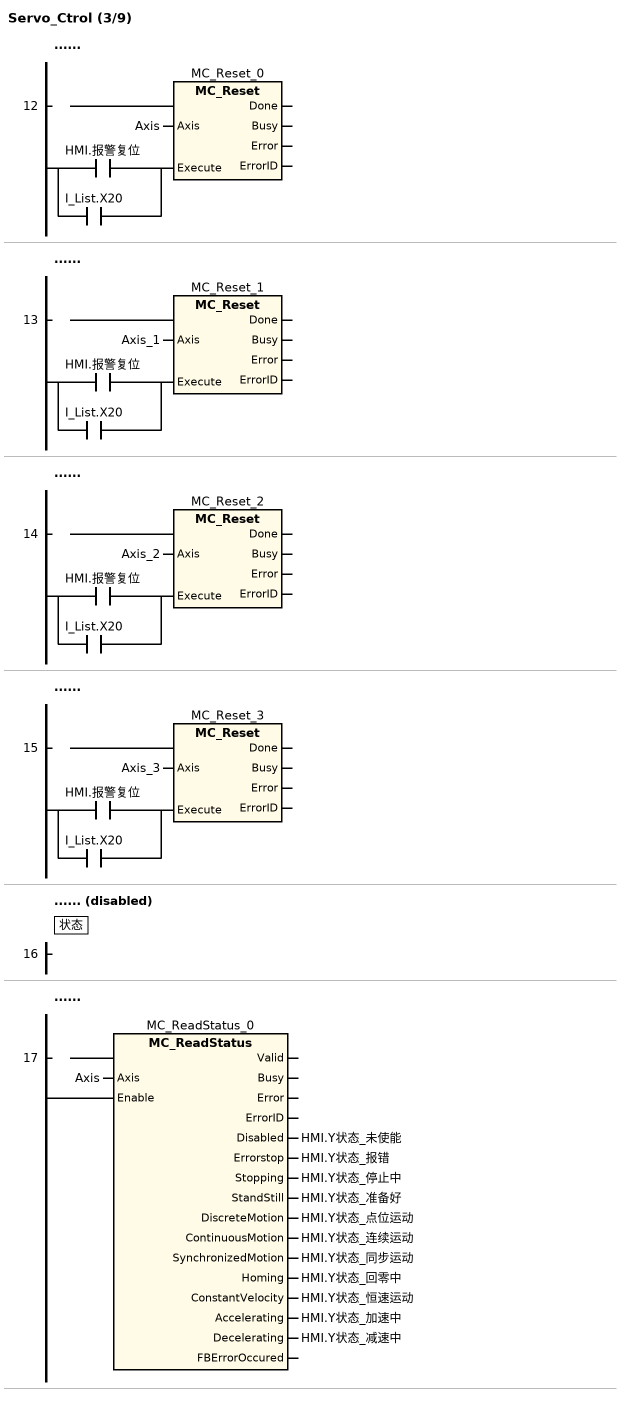
// NETWORK 12: ......
MC_Reset_0(Axis := Axis, Execute := HMI.报警复位 OR I_List.X20); // MC_Reset

// NETWORK 13: ......
MC_Reset_1(Axis := Axis_1, Execute := HMI.报警复位 OR I_List.X20); // MC_Reset

// NETWORK 14: ......
MC_Reset_2(Axis := Axis_2, Execute := HMI.报警复位 OR I_List.X20); // MC_Reset

// NETWORK 15: ......
MC_Reset_3(Axis := Axis_3, Execute := HMI.报警复位 OR I_List.X20); // MC_Reset

// NETWORK 16: ...... (disabled)
// label: 状态

// NETWORK 17: ......
MC_ReadStatus_0(
    Axis := Axis,
    Enable := TRUE,
    Disabled => HMI.Y状态_未使能,
    Errorstop => HMI.Y状态_报错,
    Stopping => HMI.Y状态_停止中,
    StandStill => HMI.Y状态_准备好,
    DiscreteMotion => HMI.Y状态_点位运动,
    ContinuousMotion => HMI.Y状态_连续运动,
    SynchronizedMotion => HMI.Y状态_同步运动,
    Homing => HMI.Y状态_回零中,
    ConstantVelocity => HMI.Y状态_恒速运动,
    Accelerating => HMI.Y状态_加速中,
    Decelerating => HMI.Y状态_减速中); // MC_ReadStatus

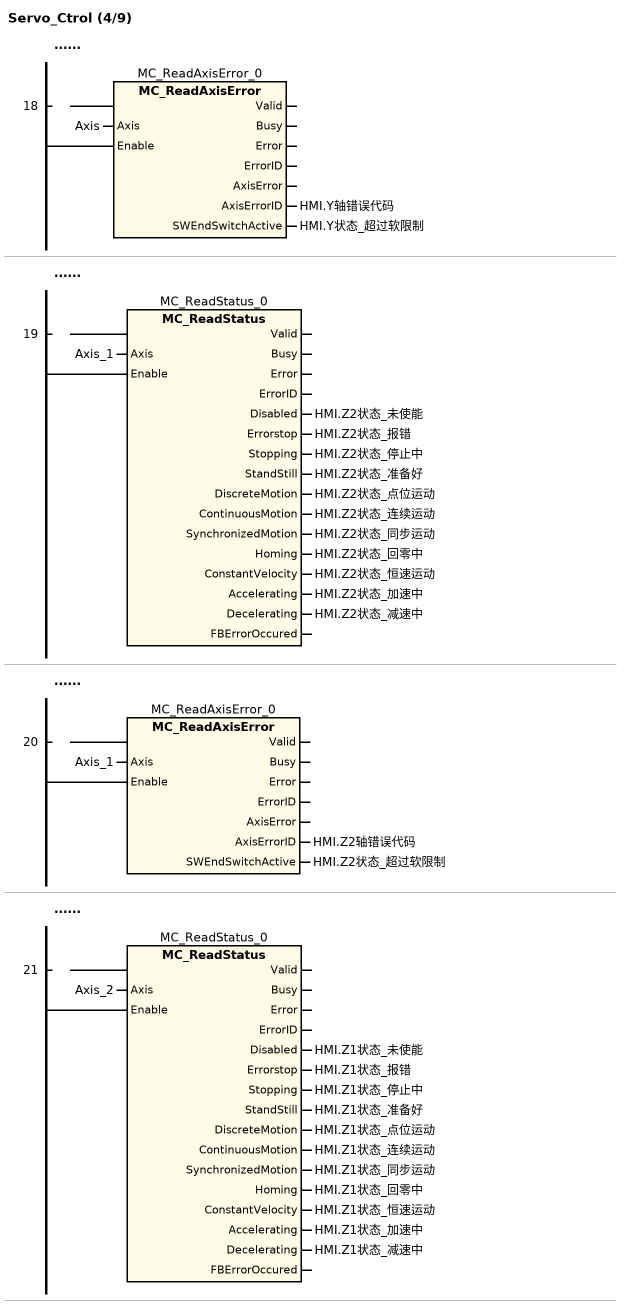
// NETWORK 18: ......
MC_ReadAxisError_0(
    Axis := Axis,
    Enable := TRUE,
    AxisErrorID => HMI.Y轴错误代码,
    SWEndSwitchActive => HMI.Y状态_超过软限制); // MC_ReadAxisError

// NETWORK 19: ......
MC_ReadStatus_0(
    Axis := Axis_1,
    Enable := TRUE,
    Disabled => HMI.Z2状态_未使能,
    Errorstop => HMI.Z2状态_报错,
    Stopping => HMI.Z2状态_停止中,
    StandStill => HMI.Z2状态_准备好,
    DiscreteMotion => HMI.Z2状态_点位运动,
    ContinuousMotion => HMI.Z2状态_连续运动,
    SynchronizedMotion => HMI.Z2状态_同步运动,
    Homing => HMI.Z2状态_回零中,
    ConstantVelocity => HMI.Z2状态_恒速运动,
    Accelerating => HMI.Z2状态_加速中,
    Decelerating => HMI.Z2状态_减速中); // MC_ReadStatus

// NETWORK 20: ......
MC_ReadAxisError_0(
    Axis := Axis_1,
    Enable := TRUE,
    AxisErrorID => HMI.Z2轴错误代码,
    SWEndSwitchActive => HMI.Z2状态_超过软限制); // MC_ReadAxisError

// NETWORK 21: ......
MC_ReadStatus_0(
    Axis := Axis_2,
    Enable := TRUE,
    Disabled => HMI.Z1状态_未使能,
    Errorstop => HMI.Z1状态_报错,
    Stopping => HMI.Z1状态_停止中,
    StandStill => HMI.Z1状态_准备好,
    DiscreteMotion => HMI.Z1状态_点位运动,
    ContinuousMotion => HMI.Z1状态_连续运动,
    SynchronizedMotion => HMI.Z1状态_同步运动,
    Homing => HMI.Z1状态_回零中,
    ConstantVelocity => HMI.Z1状态_恒速运动,
    Accelerating => HMI.Z1状态_加速中,
    Decelerating => HMI.Z1状态_减速中); // MC_ReadStatus

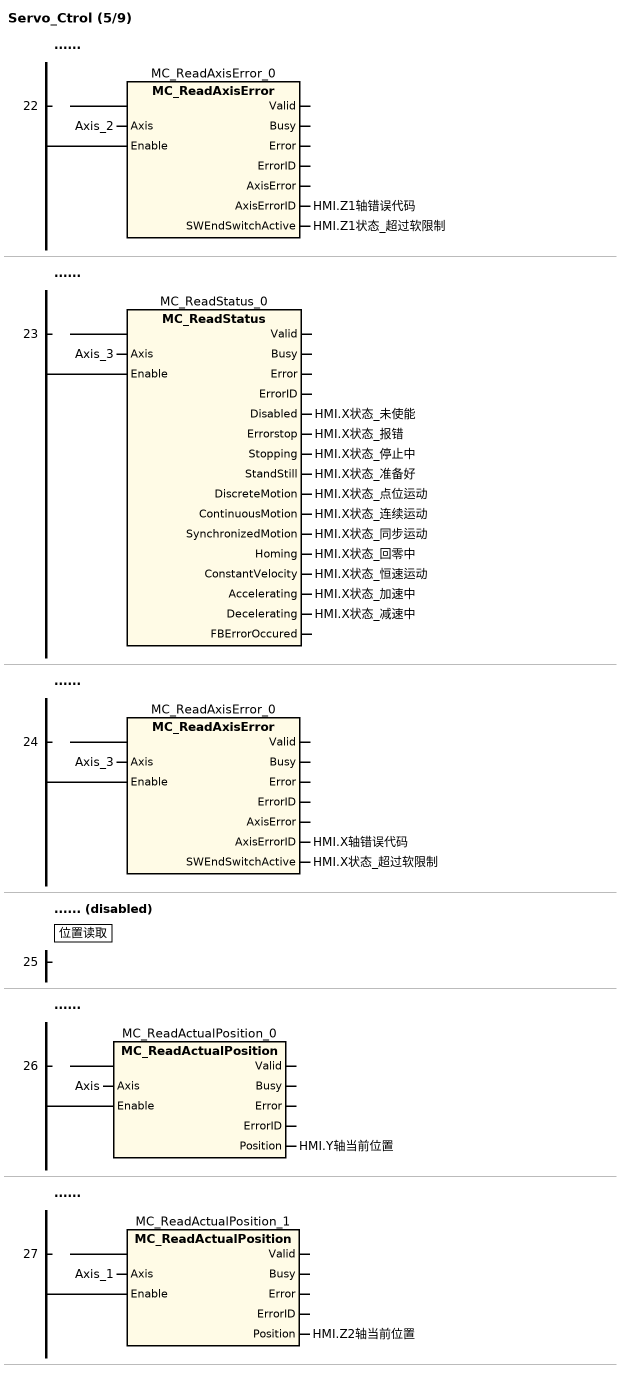
// NETWORK 22: ......
MC_ReadAxisError_0(
    Axis := Axis_2,
    Enable := TRUE,
    AxisErrorID => HMI.Z1轴错误代码,
    SWEndSwitchActive => HMI.Z1状态_超过软限制); // MC_ReadAxisError

// NETWORK 23: ......
MC_ReadStatus_0(
    Axis := Axis_3,
    Enable := TRUE,
    Disabled => HMI.X状态_未使能,
    Errorstop => HMI.X状态_报错,
    Stopping => HMI.X状态_停止中,
    StandStill => HMI.X状态_准备好,
    DiscreteMotion => HMI.X状态_点位运动,
    ContinuousMotion => HMI.X状态_连续运动,
    SynchronizedMotion => HMI.X状态_同步运动,
    Homing => HMI.X状态_回零中,
    ConstantVelocity => HMI.X状态_恒速运动,
    Accelerating => HMI.X状态_加速中,
    Decelerating => HMI.X状态_减速中); // MC_ReadStatus

// NETWORK 24: ......
MC_ReadAxisError_0(
    Axis := Axis_3,
    Enable := TRUE,
    AxisErrorID => HMI.X轴错误代码,
    SWEndSwitchActive => HMI.X状态_超过软限制); // MC_ReadAxisError

// NETWORK 25: ...... (disabled)
// label: 位置读取

// NETWORK 26: ......
MC_ReadActualPosition_0(Axis := Axis, Enable := TRUE, Position => HMI.Y轴当前位置); // MC_ReadActualPosition

// NETWORK 27: ......
MC_ReadActualPosition_1(Axis := Axis_1, Enable := TRUE, Position => HMI.Z2轴当前位置); // MC_ReadActualPosition

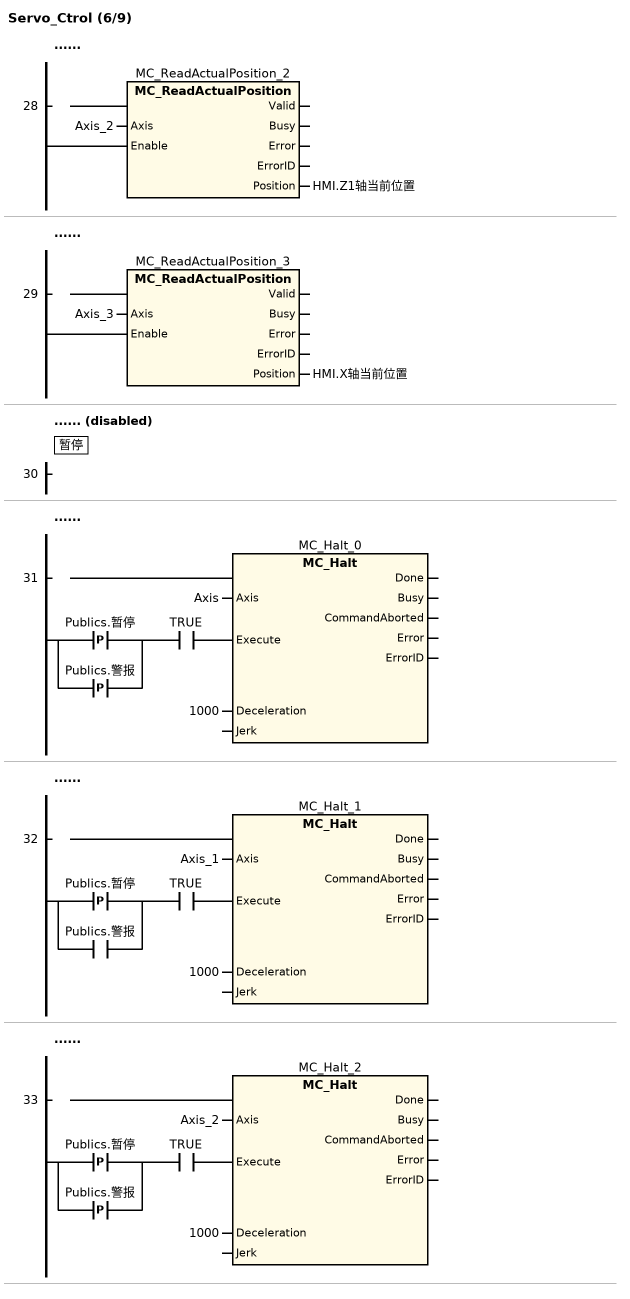
// NETWORK 28: ......
MC_ReadActualPosition_2(Axis := Axis_2, Enable := TRUE, Position => HMI.Z1轴当前位置); // MC_ReadActualPosition

// NETWORK 29: ......
MC_ReadActualPosition_3(Axis := Axis_3, Enable := TRUE, Position => HMI.X轴当前位置); // MC_ReadActualPosition

// NETWORK 30: ...... (disabled)
// label: 暂停

// NETWORK 31: ......
_rt1(CLK := Publics.暂停);
_rt2(CLK := Publics.警报);
MC_Halt_0(Axis := Axis, Execute := (_rt1.Q OR _rt2.Q) AND TRUE, Deceleration := 1000); // MC_Halt

// NETWORK 32: ......
_rt3(CLK := Publics.暂停);
MC_Halt_1(Axis := Axis_1, Execute := (_rt3.Q OR Publics.警报) AND TRUE, Deceleration := 1000); // MC_Halt

// NETWORK 33: ......
_rt4(CLK := Publics.暂停);
_rt5(CLK := Publics.警报);
MC_Halt_2(Axis := Axis_2, Execute := (_rt4.Q OR _rt5.Q) AND TRUE, Deceleration := 1000); // MC_Halt

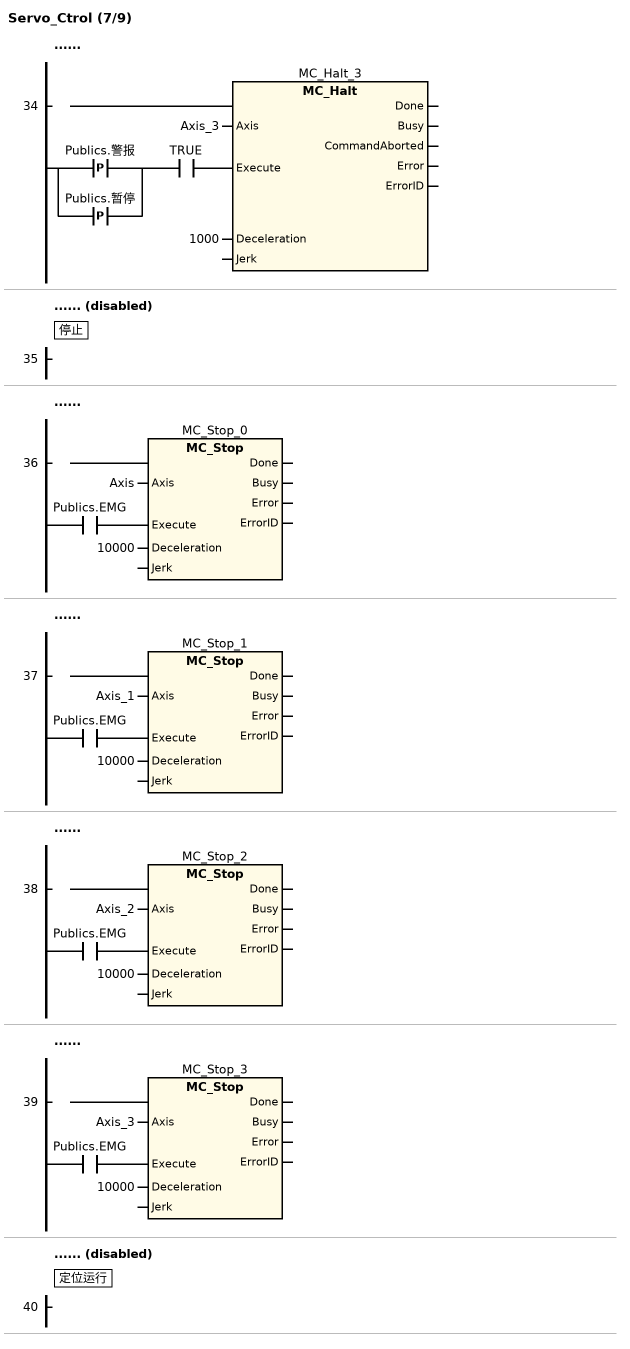
// NETWORK 34: ......
_rt6(CLK := Publics.警报);
_rt7(CLK := Publics.暂停);
MC_Halt_3(Axis := Axis_3, Execute := (_rt6.Q OR _rt7.Q) AND TRUE, Deceleration := 1000); // MC_Halt

// NETWORK 35: ...... (disabled)
// label: 停止

// NETWORK 36: ......
MC_Stop_0(Axis := Axis, Execute := Publics.EMG, Deceleration := 10000); // MC_Stop

// NETWORK 37: ......
MC_Stop_1(Axis := Axis_1, Execute := Publics.EMG, Deceleration := 10000); // MC_Stop

// NETWORK 38: ......
MC_Stop_2(Axis := Axis_2, Execute := Publics.EMG, Deceleration := 10000); // MC_Stop

// NETWORK 39: ......
MC_Stop_3(Axis := Axis_3, Execute := Publics.EMG, Deceleration := 10000); // MC_Stop

// NETWORK 40: ...... (disabled)
// label: 定位运行

